# B&R Automation Studio project TD52 (part 92)

### sPLC.var - SAFETY PLC variables
```iecst
VAR
	bSafeIN_ECW_PumpsOFF : BOOL := FALSE; (*To SafetyPLC - No engine cooling water pump is running*)
	bSafeIN_EO_PumpsOFF : BOOL := FALSE; (*To SafetyPLC - No engine oil pump is running*)
	bSafeIN_ERV_ColdCountry : BOOL := FALSE; (*To SafetyPLC - Cold country mode is active*)
	bSafeIN_ERV_Lou_PC_CL : BOOL := FALSE; (*To SafetyPLC - Plausibility check for closing the louvres*)
	bSafeIN_ERV_Lou_PC_OP : BOOL := FALSE; (*To SafetyPLC - Plausibility check for opening the louvres*)
	bSafeIN_Reset_sPLC : BOOL := FALSE; (*To SafetyPLC - RESET - Release sDOs - Reset IO card failures*)
	bSafeModuleOK_101 : BOOL := FALSE; (*Safe communication channel - Node 101 OK*)
	bSafeModuleOK_102 : BOOL := FALSE; (*Safe communication channel - Node 102 OK*)
	bSafeModuleOK_103 : BOOL := FALSE; (*Safe communication channel - Node 103 OK*)
	bSafeModuleOK_104 : BOOL := FALSE; (*Safe communication channel - Node 104 OK*)
	bSafeModuleOK_105 : BOOL := FALSE; (*Safe communication channel - Node 105 OK*)
	bSafeModuleOK_201 : BOOL := FALSE; (*Safe communication channel - Node 201 OK*)
	bSafeModuleOK_202 : BOOL := FALSE; (*Safe communication channel - Node 202 OK*)
	bSafeModuleOK_203 : BOOL := FALSE; (*Safe communication channel - Node 203 OK*)
	bSafeModuleOK_204 : BOOL := FALSE; (*Safe communication channel - Node 204 OK*)
	bSafeModuleOK_205 : BOOL := FALSE; (*Safe communication channel - Node 205 OK*)
	bSafeModuleOK_206 : BOOL := FALSE; (*Safe communication channel - Node 206 OK*)
	bSafeModuleOK_207 : BOOL := FALSE; (*Safe communication channel - Node 207 OK*)
	bSafeModuleOK_208 : BOOL := FALSE; (*Safe communication channel - Node 208 OK*)
	bSafeModuleOK_209 : BOOL := FALSE; (*Safe communication channel - Node 209 OK*)
	bSafeModuleOK_210 : BOOL := FALSE; (*Safe communication channel - Node 210 OK*)
	bSafeModuleOK_300 : BOOL := FALSE; (*Safe communication channel - Node 300 OK*)
	bSafeModuleOK_301 : BOOL := FALSE; (*Safe communication channel - Node 301 OK*)
	bSafeOUT_F01_N_DiffOK : BOOL := FALSE; (*From SafetyPLC - Function 01 - Speed difference OK*)
	bSafeOUT_F01_N_Nom90 : BOOL := FALSE; (*From SafetyPLC - Function 01 - Actual engine speed >= 90% of nominal speed*)
	bSafeOUT_F01_OK : BOOL := FALSE; (*From SafetyPLC - Function 01 - Speed measurement OK*)
	bSafeOUT_F02_OK : BOOL := FALSE; (*From SafetyPLC - Function 02 - Ignition is operating*)
	bSafeOUT_F02_OK_PC : BOOL := FALSE; (*From SafetyPLC - Function 02 - Ignition plausibility check - OK*)
	bSafeOUT_F03_OK : BOOL := FALSE; (*From SafetyPLC - Function 03 - Oil pressure MIN OK*)
	bSafeOUT_F03_Pr_EO_DiffOK : BOOL := FALSE; (*From SafetyPLC - Function 03 - Oil pressure difference OK*)
	bSafeOUT_F04_OK : BOOL := FALSE; (*From SafetyPLC - Function 04 - Oil pressure MAX OK*)
	bSafeOUT_F05_OK : BOOL := FALSE; (*From SafetyPLC - Function 05 - Engine cooling water pressure MIN OK*)
	bSafeOUT_F05_Pr_ECW_DiffOK : BOOL := FALSE; (*From SafetyPLC - Function 05 - Engine cooling water pressure difference OK*)
	bSafeOUT_F06_OK : BOOL := FALSE; (*From SafetyPLC - Function 06 - Engine cooling water pressure MAX OK*)
	bSafeOUT_F07_GCB_RUC : BOOL := FALSE; (*From SafetyPLC - Function 07 - GCB - Release undervoltage coil OK*)
	bSafeOUT_F07_GCB_RUC_PS : BOOL := FALSE; (*From SafetyPLC - Function 07 - GCB - Release undervoltage coil OK - Physical state*)
	bSafeOUT_F07_OK : BOOL := FALSE; (*From SafetyPLC - Function 07 - Grid disconnection OK*)
	bSafeOUT_F07_Rel_Sync_Load : BOOL := FALSE; (*From SafetyPLC - Function 07 - Release synchronizing and load OK*)
	bSafeOUT_F07_Rel_Sync_Load_PS : BOOL := FALSE; (*From SafetyPLC - Function 07 - Release synchronizing and load - Physical state*)
	bSafeOUT_F08_GenPrctTrip_OK : BOOL := FALSE; (*From SafetyPLC - Function 08 - Generator protection trip OK*)
	bSafeOUT_F08_OlShortCirc_OK : BOOL := FALSE; (*From SafetyPLC - Function 08 - Generator overload/short circuit OK*)
	bSafeOUT_F09_Cust_OK : BOOL := FALSE; (*From SafetyPLC - Function 09 - Room ventilation operating*)
	bSafeOUT_F09_Cust_OK_PC : BOOL := FALSE; (*From SafetyPLC - Function 09 - Room ventilation plausibility check OK*)
	bSafeOUT_F09_DI_ERV_Cust : BOOL := FALSE; (*From SafetyPLC - Function 09 - Room ventilation operating - Digital input*)
	bSafeOUT_F09_Door_OK : BOOL := FALSE; (*From SafetyPLC - Function 09 - Doors closed*)
	bSafeOUT_F09_ERV_PC_Forced : BOOL := FALSE; (*From SafetyPLC - Function 09 - Forced ERV plausibility checks*)
	bSafeOUT_F09_INL1_Fan_OK : BOOL := FALSE; (*From SafetyPLC - Function 09 - Group 1 - Inlet air fan operating*)
	bSafeOUT_F09_INL1_Fan_OK_PC : BOOL := FALSE; (*From SafetyPLC - Function 09 - Group 1 - Inlet air fan plausibility check OK*)
	bSafeOUT_F09_INL1_Lou_OK : BOOL := FALSE; (*From SafetyPLC - Function 09 - Group 1 - Inlet air louvre OK*)
	bSafeOUT_F09_INL1_Lou_OK_PC : BOOL := FALSE; (*From SafetyPLC - Function 09 - Group 1 - Inlet air louvre plausibility check OK*)
	bSafeOUT_F09_INL2_Fan_OK : BOOL := FALSE; (*From SafetyPLC - Function 09 - Group 2 - Inlet air fan operating*)
	bSafeOUT_F09_INL2_Fan_OK_PC : BOOL := FALSE; (*From SafetyPLC - Function 09 - Group 2 - Inlet air fan plausibility check OK*)
	bSafeOUT_F09_INL2_Lou_OK : BOOL := FALSE; (*From SafetyPLC - Function 09 - Group 2 - Inlet air louvre OK*)
	bSafeOUT_F09_INL2_Lou_OK_PC : BOOL := FALSE; (*From SafetyPLC - Function 09 - Group 2 - Inlet air louvre plausibility check OK*)
	bSafeOUT_F09_INL3_Fan_OK : BOOL := FALSE; (*From SafetyPLC - Function 09 - Group 3 - Inlet air fan operating*)
	bSafeOUT_F09_INL3_Fan_OK_PC : BOOL := FALSE; (*From SafetyPLC - Function 09 - Group 3 - Inlet air fan plausibility check OK*)
	bSafeOUT_F09_INL3_Lou_OK : BOOL := FALSE; (*From SafetyPLC - Function 09 - Group 3 - Inlet air louvre OK*)
	bSafeOUT_F09_INL3_Lou_OK_PC : BOOL := FALSE; (*From SafetyPLC - Function 09 - Group 3 - Inlet air louvre plausibility check OK*)
	bSafeOUT_F09_INL4_Fan_OK : BOOL := FALSE; (*From SafetyPLC - Function 09 - Group 4 - Inlet air fan operating*)
	bSafeOUT_F09_INL4_Fan_OK_PC : BOOL := FALSE; (*From SafetyPLC - Function 09 - Group 4 - Inlet air fan plausibility check OK*)
	bSafeOUT_F09_INL4_Lou_OK : BOOL := FALSE; (*From SafetyPLC - Function 09 - Group 4 - Inlet air louvre OK*)
	bSafeOUT_F09_INL4_Lou_OK_PC : BOOL := FALSE; (*From SafetyPLC - Function 09 - Group 4 - Inlet air louvre plausibility check OK*)
	bSafeOUT_F09_INL5_Fan_OK : BOOL := FALSE; (*From SafetyPLC - Function 09 - Group 5 - Inlet air fan operating*)
	bSafeOUT_F09_INL5_Fan_OK_PC : BOOL := FALSE; (*From SafetyPLC - Function 09 - Group 5 - Inlet air fan plausibility check OK*)
	bSafeOUT_F09_INL5_Lou_OK : BOOL := FALSE; (*From SafetyPLC - Function 09 - Group 5 - Inlet air louvre OK*)
	bSafeOUT_F09_INL5_Lou_OK_PC : BOOL := FALSE; (*From SafetyPLC - Function 09 - Group 5 - Inlet air louvre plausibility check OK*)
	bSafeOUT_F09_INL6_Fan_OK : BOOL := FALSE; (*From SafetyPLC - Function 09 - Group 6 - Inlet air fan operating*)
	bSafeOUT_F09_INL6_Fan_OK_PC : BOOL := FALSE; (*From SafetyPLC - Function 09 - Group 6 - Inlet air fan plausibility check OK*)
	bSafeOUT_F09_INL6_Lou_OK : BOOL := FALSE; (*From SafetyPLC - Function 09 - Group 6 - Inlet air louvre OK*)
	bSafeOUT_F09_INL6_Lou_OK_PC : BOOL := FALSE; (*From SafetyPLC - Function 09 - Group 6 - Inlet air louvre plausibility check OK*)
	bSafeOUT_F09_OTL1_Lou_OK : BOOL := FALSE; (*From SafetyPLC - Function 09 - Group 1 - Outlet air louvre OK*)
	bSafeOUT_F09_OTL1_Lou_OK_PC : BOOL := FALSE; (*From SafetyPLC - Function 09 - Group 1 - Outlet air louvre plausibility check OK*)
	bSafeOUT_F09_OTL2_Lou_OK : BOOL := FALSE; (*From SafetyPLC - Function 09 - Group 2 - Outlet air louvre OK*)
	bSafeOUT_F09_OTL2_Lou_OK_PC : BOOL := FALSE; (*From SafetyPLC - Function 09 - Group 2 - Outlet air louvre plausibility check OK*)
	bSafeOUT_F09_OTL3_Lou_OK : BOOL := FALSE; (*From SafetyPLC - Function 09 - Group 3 - Outlet air louvre OK*)
	bSafeOUT_F09_OTL3_Lou_OK_PC : BOOL := FALSE; (*From SafetyPLC - Function 09 - Group 3 - Outlet air louvre plausibility check OK*)
	bSafeOUT_F09_OTL4_Lou_OK : BOOL := FALSE; (*From SafetyPLC - Function 09 - Group 4 - Outlet air louvre OK*)
	bSafeOUT_F09_OTL4_Lou_OK_PC : BOOL := FALSE; (*From SafetyPLC - Function 09 - Group 4 - Outlet air louvre plausibility check OK*)
	bSafeOUT_F09_OTL5_Lou_OK : BOOL := FALSE; (*From SafetyPLC - Function 09 - Group 5 - Outlet air louvre OK*)
	bSafeOUT_F09_OTL5_Lou_OK_PC : BOOL := FALSE; (*From SafetyPLC - Function 09 - Group 5 - Outlet air louvre plausibility check OK*)
	bSafeOUT_F09_OTL6_Lou_OK : BOOL := FALSE; (*From SafetyPLC - Function 09 - Group 6 - Outlet air louvre OK*)
	bSafeOUT_F09_OTL6_Lou_OK_PC : BOOL := FALSE; (*From SafetyPLC - Function 09 - Group 6 - Outlet air louvre plausibility check OK*)
	bSafeOUT_F10_DO_EmStop : BOOL := FALSE; (*From SafetyPLC - Function 10 - DO Emergency stop signalling*)
	bSafeOUT_F10_DO_EmStop_PS : BOOL := FALSE; (*From SafetyPLC - Function 10 - DO Emergency stop signalling - Physical state*)
	bSafeOUT_F10_EmStop_M_OK : BOOL := FALSE; (*From SafetyPLC - Function 10 - Emergency stop push button - Module interface panel*)
	bSafeOUT_F10_EmStop_OK : BOOL := FALSE; (*From SafetyPLC - Function 10 - Emergency stop push button*)
	bSafeOUT_F10_SafetyLoop_EmStop : BOOL := FALSE; (*From SafetyPLC - Function 10 - Safety loop - Emergency stop push button OK*)
	bSafeOUT_F11_SafetyLoop_A1_OK : BOOL := FALSE; (*From SafetyPLC - Function 11 - Safety loop 1 - module control panel OK*)
	bSafeOUT_F11_SafetyLoop_A2_OK : BOOL := FALSE; (*From SafetyPLC - Function 11 - Safety loop 2 - module control panel OK*)
	bSafeOUT_F11_SafetyLoop_M_OK : BOOL := FALSE; (*From SafetyPLC - Function 11 - Safety loop - module interface panel OK*)
	bSafeOUT_F12_DCGA_OK : BOOL := FALSE; (*From SafetyPLC - Function 12 - Gas supply interruption OK - DCGA (Decentral gas addition)*)
	bSafeOUT_F12_DCGA_SD_Dem : BOOL := FALSE; (*From SafetyPLC - Function 12 - Demand gas safety device - DCGA*)
	bSafeOUT_F12_DCGA_SD_Dem_PS : BOOL := FALSE; (*From SafetyPLC - Function 12 - Demand gas safety device - DCGA - Physical state*)
	bSafeOUT_F12_DI_DCGA_SafeDevOK : BOOL := FALSE; (*From SafetyPLC - Function 12 - Digital Input - Gas safety device OK - DCGA*)
	bSafeOUT_F12_DI_GT1_SafeDevOK : BOOL := FALSE; (*From SafetyPLC - Function 12 - Digital Input - Gas safety device OK - Gastrain 1*)
	bSafeOUT_F12_DI_GT2_SafeDevOK : BOOL := FALSE; (*From SafetyPLC - Function 12 - Digital Input - Gas safety device OK - Gastrain 2*)
	bSafeOUT_F12_DI_GT3_SafeDevOK : BOOL := FALSE; (*From SafetyPLC - Function 12 - Digital Input - Gas safety device OK - Gastrain 3*)
	bSafeOUT_F12_DI_GT4_SafeDevOK : BOOL := FALSE; (*From SafetyPLC - Function 12 - Digital Input - Gas safety device OK - Gastrain 4*)
	bSafeOUT_F12_GT1_OK : BOOL := FALSE; (*From SafetyPLC - Function 12 - Gas supply interruption OK - Gas train 1*)
	bSafeOUT_F12_GT1_SD_Dem : BOOL := FALSE; (*From SafetyPLC - Function 12 - Demand gas safety device - Gastrain 1*)
	bSafeOUT_F12_GT1_SD_Dem_PS : BOOL := FALSE; (*From SafetyPLC - Function 12 - Demand gas safety device - Gastrain 1 - Physical state*)
	bSafeOUT_F12_GT2_OK : BOOL := FALSE; (*From SafetyPLC - Function 12 - Gas supply interruption OK - Gas train 2*)
	bSafeOUT_F12_GT2_SD_Dem : BOOL := FALSE; (*From SafetyPLC - Function 12 - Demand gas safety device - Gastrain 2*)
	bSafeOUT_F12_GT2_SD_Dem_PS : BOOL := FALSE; (*From SafetyPLC - Function 12 - Demand gas safety device - Gastrain 2 - Physical state*)
	bSafeOUT_F12_GT3_OK : BOOL := FALSE; (*From SafetyPLC - Function 12 - Gas supply interruption OK - Gas train 3*)
	bSafeOUT_F12_GT3_SD_Dem : BOOL := FALSE; (*From SafetyPLC - Function 12 - Demand gas safety device - Gastrain 3*)
	bSafeOUT_F12_GT3_SD_Dem_PS : BOOL := FALSE; (*From SafetyPLC - Function 12 - Demand gas safety device - Gastrain 3 - Physical state*)
	bSafeOUT_F12_GT4_OK : BOOL := FALSE; (*From SafetyPLC - Function 12 - Gas supply interruption OK - Gas train 4*)
	bSafeOUT_F12_GT4_SD_Dem : BOOL := FALSE; (*From SafetyPLC - Function 12 - Demand gas safety device - Gastrain 4*)
	bSafeOUT_F12_GT4_SD_Dem_PS : BOOL := FALSE; (*From SafetyPLC - Function 12 - Demand gas safety device - Gastrain 4 - Physical state*)
	bSafeOUT_F12_Rel_GV1 : BOOL := FALSE; (*From SafetyPLC - Function 12 - Gas valves from gas train 1 released*)
	bSafeOUT_F12_Rel_GV1a_PS : BOOL := FALSE; (*From SafetyPLC - Function 12 - Gas valve 1a - Physical state*)
	bSafeOUT_F12_Rel_GV1b_PS : BOOL := FALSE; (*From SafetyPLC - Function 12 - Gas valve 1b - Physical state*)
	bSafeOUT_F12_Rel_GV2 : BOOL := FALSE; (*From SafetyPLC - Function 12 - Gas valves from gas train 2 released*)
	bSafeOUT_F12_Rel_GV2a_PS : BOOL := FALSE; (*From SafetyPLC - Function 12 - Gas valve 2a - Physical state*)
	bSafeOUT_F12_Rel_GV2b_PS : BOOL := FALSE; (*From SafetyPLC - Function 12 - Gas valve 2b - Physical state*)
	bSafeOUT_F12_Rel_GV3 : BOOL := FALSE; (*From SafetyPLC - Function 12 - Gas valves from gas train 3 released*)
	bSafeOUT_F12_Rel_GV3a_PS : BOOL := FALSE; (*From SafetyPLC - Function 12 - Gas valve 3a - Physical state*)
	bSafeOUT_F12_Rel_GV3b_PS : BOOL := FALSE; (*From SafetyPLC - Function 12 - Gas valve 3b - Physical state*)
	bSafeOUT_F12_Rel_GV4 : BOOL := FALSE; (*From SafetyPLC - Function 12 - Gas valves from gas train 4 released*)
	bSafeOUT_F12_Rel_GV4a_PS : BOOL := FALSE; (*From SafetyPLC - Function 12 - Gas valve 4a - Physical state*)
	bSafeOUT_F12_Rel_GV4b_PS : BOOL := FALSE; (*From SafetyPLC - Function 12 - Gas valve 4b - Physical state*)
	bSafeOUT_F12_Rel_GVa_DCGA_PS : BOOL := FALSE; (*From SafetyPLC - Function 12 - Gas valve a for DCGA - Physical state*)
	bSafeOUT_F12_Rel_GVb_DCGA_PS : BOOL := FALSE; (*From SafetyPLC - Function 12 - Gas valve b for DCGA - Physical state*)
	bSafeOUT_F12_Rel_GV_DCGA : BOOL := FALSE; (*From SafetyPLC - Function 12 - Gas valves from DCGA released*)
	bSafeOUT_F16_DI_ScavFlapClosed : BOOL := FALSE; (*From SafetyPLC - Function 20 - Scavenging flap closed OK*)
	bSafeOUT_F16_ScavFlapPos_OK : BOOL := FALSE; (*From SafetyPLC - Function 20 - Scavenging flap position OK*)
	bSafeOUT_F16_ScavFlapPos_OK_PC : BOOL := FALSE; (*From SafetyPLC - Function 20 - Scavenging flap position - plausibility check  OK*)
	bSafeOUT_F16_TS_ScavFlap_OK : BOOL := FALSE; (*From SafetyPLC - Function 20 - Scavenging flap temperature switch  OK*)
	bSafeOUT_F17_Purge_OK : BOOL := FALSE; (*From SafetyPLC - Function 17 - Purge state OK*)
	bSafeOUT_F20_FS_HWHT_Lo_DI : BOOL := FALSE; (*From SafetyPLC - Function 20 - High temperature heating water flow minimum - DI OK*)
	bSafeOUT_F20_FS_HWHT_Lo_OK : BOOL := FALSE; (*From SafetyPLC - Function 20 - High temperature heating water flow minimum OK*)
	bSafeOUT_F20_FS_HWHT_Lo_OK_PC : BOOL := FALSE; (*From SafetyPLC - Function 20 - High temperature heating water flow minimum - plausibility check OK*)
	bSafeOUT_F20_FS_HWLT_Lo_DI : BOOL := FALSE; (*From SafetyPLC - Function 20 - Low temperature heating water flow minimum - DI OK*)
	bSafeOUT_F20_FS_HWLT_Lo_OK : BOOL := FALSE; (*From SafetyPLC - Function 20 - Low temperature heating water flow minimum OK*)
	bSafeOUT_F20_FS_HWLT_Lo_OK_PC : BOOL := FALSE; (*From SafetyPLC - Function 20 - Low temperature heating water flow minimum - plausibility check OK*)
	bSafeOUT_F20_HWcirc_Cust_OK : BOOL := FALSE; (*From SafetyPLC - Function 20 - Customer heating water circuit OK*)
	bSafeOUT_F20_LS_HWHT_Lo_OK : BOOL := FALSE; (*From SafetyPLC - Function 20 - High temperature heating water level minimum OK*)
	bSafeOUT_F20_LS_HWLT_Lo_OK : BOOL := FALSE; (*From SafetyPLC - Function 20 - Low temperature heating water level minimum OK*)
	bSafeOUT_F20_PS1_HWHT_Hi_OK : BOOL := FALSE; (*From SafetyPLC - Function 20 - High temperature heating water pressure 1 maximum OK*)
	bSafeOUT_F20_PS1_HWHT_Lo_DI : BOOL := FALSE; (*From SafetyPLC - Function 20 - High temperature heating water pressure 1 minimum - DI OK*)
	bSafeOUT_F20_PS1_HWHT_Lo_OK : BOOL := FALSE; (*From SafetyPLC - Function 20 - High temperature heating water pressure 1 minimum OK*)
	bSafeOUT_F20_PS1_HWLT_Hi_OK : BOOL := FALSE; (*From SafetyPLC - Function 20 - Low temperature heating water pressure 1 maximum OK*)
	bSafeOUT_F20_PS1_HWLT_Lo_DI : BOOL := FALSE; (*From SafetyPLC - Function 20 - Low temperature heating water pressure 1 minimum - DI OK*)
	bSafeOUT_F20_PS1_HWLT_Lo_OK : BOOL := FALSE; (*From SafetyPLC - Function 20 - Low temperature heating water pressure 1 minimum OK*)
	bSafeOUT_F20_PS2_HWHT_Hi_OK : BOOL := FALSE; (*From SafetyPLC - Function 20 - High temperature heating water pressure 2 maximum OK*)
	bSafeOUT_F20_PS2_HWHT_Lo_DI : BOOL := FALSE; (*From SafetyPLC - Function 20 - High temperature heating water pressure 2 minimum - DI OK*)
	bSafeOUT_F20_PS2_HWHT_Lo_OK : BOOL := FALSE; (*From SafetyPLC - Function 20 - High temperature heating water pressure 2 minimum OK*)
	bSafeOUT_F20_PS2_HWLT_Hi_OK : BOOL := FALSE; (*From SafetyPLC - Function 20 - Low temperature heating water pressure 2 maximum OK*)
	bSafeOUT_F20_PS2_HWLT_Lo_DI : BOOL := FALSE; (*From SafetyPLC - Function 20 - Low temperature heating water pressure 2 minimum - DI OK*)
	bSafeOUT_F20_PS2_HWLT_Lo_OK : BOOL := FALSE; (*From SafetyPLC - Function 20 - Low temperature heating water pressure 2 minimum OK*)
	bSafeOUT_F20_TS1_HWHT_Hi_OK : BOOL := FALSE; (*From SafetyPLC - Function 20 - High temperature heating water temperature 1 maximum OK*)
	bSafeOUT_F20_TS1_HWLT_Hi_OK : BOOL := FALSE; (*From SafetyPLC - Function 20 - Low temperature heating water temperature 1 maximum OK*)
	bSafeOUT_F20_TS2_HWHT_Hi_OK : BOOL := FALSE; (*From SafetyPLC - Function 20 - High temperature heating water temperature 2 maximum OK*)
	bSafeOUT_F20_TS2_HWLT_Hi_OK : BOOL := FALSE; (*From SafetyPLC - Function 20 - Low temperature heating water temperature 2 maximum OK*)
	bSafeOUT_F21_Pr_EG_Hi_OK : BOOL := FALSE; (*From SafetyPLC - Function 20 - Exhaust gas backpressure high OK*)
	bSafeOUT_F99_Rel_SF_OK : BOOL := FALSE; (*From SafetyPLC - Function 99 - Release safety functions OK*)
	bSafeOUT_F99_Rel_SF_OK_A_PS : BOOL := FALSE; (*From SafetyPLC - Function 99 - Release safety functions - Module control panel - Physical state*)
	bSafeOUT_F99_Rel_SF_OK_M_PS : BOOL := FALSE; (*From SafetyPLC - Function 99 - Release safety functions - Module interface panel - Physical state*)
	bSafeOUT_F99_SafetyLoop_Eng : BOOL := FALSE; (*From SafetyPLC - Function 10 - Safety loop - Engine OK*)
	iParaRead_sPLC : ARRAY[0..29] OF UINT := [30(0)]; (*Read Parameter from SafetyPLC*)
	iSafeIN_Eng_Motortype : INT := 0; (*To SafetyPLC - Para: Motortype*)
	iSafeIN_N_EngAct : INT := 0; (*To SafetyPLC - Actual engine speed [rpm]*)
	iSafeIN_N_EngNom : INT := 0; (*To SafetyPLC - Para: Engine nominal speed [rpm]*)
	iSafeOUT_F01_N_EngAct : DINT := 0; (*From SafetyPLC - Function 01 - Actual engine speed [rpm]*)
	iSafeOUT_F01_N_EngAct_Diff : DINT := 0; (*From SafetyPLC - Function 01 - Speed difference [rpm]*)
	iSafeOUT_F01_N_Nom90_10s_ET : DINT := 0; (*From SafetyPLC - Function 01 - Speed >= 90% of nominal speed - Elipsed time*)
	iSafeOUT_F01_SDC_30s_ET : DINT := 0; (*From SafetyPLC - Function 01 - Speed difference check - Elipsed time*)
	iSafeOUT_F01_Standstill_1m_ET : DINT := 0; (*From SafetyPLC - Function 01 - Speed < 80rpm - Elipsed time*)
	iSafeOUT_F03_Pr_EO : DINT := 0; (*From SafetyPLC - Function 03 - Actual oil pressure at last lubrication point [mbar]*)
	iSafeOUT_F03_Pr_EO_Diff : DINT := 0; (*From SafetyPLC - Function 03 - Oil pressure difference [mbar]*)
	iSafeOUT_F03_Pr_EO_Fr_1m_ET : DINT := 0; (*From SafetyPLC - Function 03 - Oil pressure frozen - Elipsed time*)
	iSafeOUT_F03_Pr_EO_Standstill : DINT := 0; (*From SafetyPLC - Function 03 - Oil pressure at last lubrication point - At standstill [mbar]*)
	iSafeOUT_F04_EO_PumpsOff_2m_ET : DINT := 0; (*From SafetyPLC - Function 04 - Oil pumps off for 120s - Elipsed time*)
	iSafeOUT_F04_Pr_EOaP : DINT := 0; (*From SafetyPLC - Function 04 - Actual oil pressure after pump [mbar]*)
	iSafeOUT_F04_Pr_EOaP_Fr_1m_ET : DINT := 0; (*From SafetyPLC - Function 04 - Oil pressure after pump frozen - Elipsed time*)
	iSafeOUT_F04_Pr_EOaP_Standstill : DINT := 0; (*From SafetyPLC - Function 04 - Oil pressure after pump - At standstill [mbar]*)
	iSafeOUT_F05_Pr_ECW : DINT := 0; (*From SafetyPLC - Function 05 - Actual engine cooling water pressure [mbar]*)
	iSafeOUT_F05_Pr_ECW_Diff : DINT := 0; (*From SafetyPLC - Function 05 - Engine cooling water pressure difference [mbar]*)
	iSafeOUT_F05_Pr_ECW_Fr_1m_ET : DINT := 0; (*From SafetyPLC - Function 05 - Engine cooling water pressure frozen - Elipsed time*)
	iSafeOUT_F06_ECW_PumpsOff_2m_ET : DINT := 0; (*From SafetyPLC - Function 06 - Engine cooling water pumps off for 120s - Elipsed time*)
	iSafeOUT_F06_Pr_ECWaP : DINT := 0; (*From SafetyPLC - Function 06 - Actual engine cooling water pressure after pump [mbar]*)
	iSafeOUT_F06_Pr_ECWaP_Fr_1m_ET : DINT := 0; (*From SafetyPLC - Function 06 - Engine cooling water pressure after pump frozen - Elipsed time*)
	iSafeOUT_F07_GCB_On_10s_ET : DINT := 0; (*From SafetyPLC - Function 07 - Generator circuit breaker ON for 10s - Elipsed time*)
	iSafeOUT_F07_GCB_On_60s_ET : DINT := 0; (*From SafetyPLC - Function 07 - Generator circuit breaker ON for 60s - Elipsed time*)
	iSafeOUT_F09_CRC : UDINT := 0; (*From SafetyPLC - Function 09 - Ventilation - CRC*)
	iSafeOUT_F09_Cust_OK_15s_ET : DINT := 0; (*From SafetyPLC - Function 09 - Room ventilation not operating - Elapsed time*)
	iSafeOUT_F09_Cust_PC_ET : DINT := 0; (*From SafetyPLC - Function 09 - Room ventilation plausibility check - Elapsed time*)
	iSafeOUT_F09_Door_OK_15s_ET : DINT := 0; (*From SafetyPLC - Function 09 - Doors not closed - Elapsed time*)
	iSafeOUT_F09_INL1_Fan_OK_1m_ET : DINT := 0; (*From SafetyPLC - Function 09 - Group 1 - Inlet air fan not operating - Elapsed time*)
	iSafeOUT_F09_INL1_Lou_OK_1m_ET : DINT := 0; (*From SafetyPLC - Function 09 - Group 1 - Inlet air louvre not OK - Elapsed time*)
	iSafeOUT_F09_INL2_Fan_OK_1m_ET : DINT := 0; (*From SafetyPLC - Function 09 - Group 2 - Inlet air fan not operating - Elapsed time*)
	iSafeOUT_F09_INL2_Lou_OK_1m_ET : DINT := 0; (*From SafetyPLC - Function 09 - Group 2 - Inlet air louvre not OK - Elapsed time*)
	iSafeOUT_F09_INL3_Fan_OK_1m_ET : DINT := 0; (*From SafetyPLC - Function 09 - Group 3 - Inlet air fan not operating - Elapsed time*)
	iSafeOUT_F09_INL3_Lou_OK_1m_ET : DINT := 0; (*From SafetyPLC - Function 09 - Group 3 - Inlet air louvre not OK - Elapsed time*)
	iSafeOUT_F09_INL4_Fan_OK_1m_ET : DINT := 0; (*From SafetyPLC - Function 09 - Group 4 - Inlet air fan not operating - Elapsed time*)
	iSafeOUT_F09_INL4_Lou_OK_1m_ET : DINT := 0; (*From SafetyPLC - Function 09 - Group 4 - Inlet air louvre not OK - Elapsed time*)
	iSafeOUT_F09_INL5_Fan_OK_1m_ET : DINT := 0; (*From SafetyPLC - Function 09 - Group 5 - Inlet air fan not operating - Elapsed time*)
	iSafeOUT_F09_INL5_Lou_OK_1m_ET : DINT := 0; (*From SafetyPLC - Function 09 - Group 5 - Inlet air louvre not OK - Elapsed time*)
	iSafeOUT_F09_INL6_Fan_OK_1m_ET : DINT := 0; (*From SafetyPLC - Function 09 - Group 6 - Inlet air fan not operating - Elapsed time*)
	iSafeOUT_F09_INL6_Lou_OK_1m_ET : DINT := 0; (*From SafetyPLC - Function 09 - Group 6 - Inlet air louvre not OK - Elapsed time*)
	iSafeOUT_F09_Nr_PC_NotDone : INT := 0; (*From SafetyPLC - Function 09 - Number of plausibility checks not performed*)
	iSafeOUT_F09_OTL1_Lou_OK_1m_ET : DINT := 0; (*From SafetyPLC - Function 09 - Group 1 - Outlet air louvre not OK - Elapsed time*)
	iSafeOUT_F09_OTL2_Lou_OK_1m_ET : DINT := 0; (*From SafetyPLC - Function 09 - Group 2 - Outlet air louvre not OK - Elapsed time*)
	iSafeOUT_F09_OTL3_Lou_OK_1m_ET : DINT := 0; (*From SafetyPLC - Function 09 - Group 3 - Outlet air louvre not OK - Elapsed time*)
	iSafeOUT_F09_OTL4_Lou_OK_1m_ET : DINT := 0; (*From SafetyPLC - Function 09 - Group 4 - Outlet air louvre not OK - Elapsed time*)
	iSafeOUT_F09_OTL5_Lou_OK_1m_ET : DINT := 0; (*From SafetyPLC - Function 09 - Group 5 - Outlet air louvre not OK - Elapsed time*)
	iSafeOUT_F09_OTL6_Lou_OK_1m_ET : DINT := 0; (*From SafetyPLC - Function 09 - Group 6 - Outlet air louvre not OK - Elapsed time*)
	iSafeOUT_F12_DCGA_LC_130s_ET : DINT := 0; (*From SafetyPLC - Function 12 - DCGA - Gas leakage check 130s - Elipsed time*)
	iSafeOUT_F12_GT1_LC_130s_ET : DINT := 0; (*From SafetyPLC - Function 12 - Gas train 1 - Gas leakage check 130s - Elipsed time*)
	iSafeOUT_F12_GT2_LC_130s_ET : DINT := 0; (*From SafetyPLC - Function 12 - Gas train 2 - Gas leakage check 130s - Elipsed time*)
	iSafeOUT_F12_GT3_LC_130s_ET : DINT := 0; (*From SafetyPLC - Function 12 - Gas train 3 - Gas leakage check 130s - Elipsed time*)
	iSafeOUT_F12_GT4_LC_130s_ET : DINT := 0; (*From SafetyPLC - Function 12 - Gas train 4 - Gas leakage check 130s - Elipsed time*)
	iSafeOUT_F12_GV_Open_60s_ET : DINT := 0; (*From SafetyPLC - Function 12 - Gas valves open for 60s - Elipsed time*)
	iSafeOUT_F16_ScavFlapPos_PC_ET : DINT := 0; (*From SafetyPLC - Function 16 - Scavenging flap position - plausibility check - Elipsed time OK*)
	iSafeOUT_F17_Vol_PurgeAir : DINT := 0; (*From SafetyPLC - Function 17 - Purge air volume [l]*)
	iSafeOUT_F20_CRC : UDINT := 0; (*From SafetyPLC - Function 20 - Heating water - CRC*)
	iSafeOUT_F20_FS_HWHT_Lo_OK_ET : DINT := 0; (*From SafetyPLC - Function 20 - High temperature heating water flow minimum - Elipsed time OK*)
	iSafeOUT_F20_FS_HWHT_Lo_PC_ET : DINT := 0; (*From SafetyPLC - Function 20 - High temperature heating water flow minimum - plausibility check - Elipsed time OK*)
	iSafeOUT_F20_FS_HWLT_Lo_OK_ET : DINT := 0; (*From SafetyPLC - Function 20 - Low temperature heating water flow minimum - Elipsed time OK*)
	iSafeOUT_F20_FS_HWLT_Lo_PC_ET : DINT := 0; (*From SafetyPLC - Function 20 - Low temperature heating water flow minimum - plausibility check - Elipsed time OK*)
	iSafeOUT_F20_PS1_HWHT_Lo_OK_ET : DINT := 0; (*From SafetyPLC - Function 20 - High temperature heating water pressure 1 minimum - Elipsed time OK*)
	iSafeOUT_F20_PS1_HWLT_Lo_OK_ET : DINT := 0; (*From SafetyPLC - Function 20 - Low temperature heating water pressure 1 minimum - Elipsed time OK*)
	iSafeOUT_F20_PS2_HWHT_Lo_OK_ET : DINT := 0; (*From SafetyPLC - Function 20 - High temperature heating water pressure 2 minimum - Elipsed time OK*)
	iSafeOUT_F20_PS2_HWLT_Lo_OK_ET : DINT := 0; (*From SafetyPLC - Function 20 - Low temperature heating water pressure 2 minimum - Elipsed time OK*)
	iSafeOUT_FwVers_sPLC : UDINT := 0; (*From SafetyPLC - Actual firmware version*)
	MM2VIS_sPLC : MM2VIS_sPLC_Struct;
	VIS2MM_sPLC : VIS2MM_sPLC_struct;
END_VAR
```

### Program Logical/EngineGeneral/GeneralEG (IEC, version 4.10.0) - general functions

#### GeneralEGCyclic.st - Cyclic code
```iecst
(*******************************************************************************
GeneralEG		general functions

This code is confidential and proprietary to the INNIO Company.
It may not be used in any form, or reproduced in any manner,
without the express written permission of the INNIO Company.
Copyright, INNIO Company, 2021

Customized modifications: -
------------------------

History:
-------
V03.99.00.00	08.02.2013 	Tinello 	Created
V04.03.00.00	20.01.2016	Tinello		Release Module if ParaSetupOk = TRUE added
V04.05.00.00	26.01.2017	Tinello		Release Module from 10s -> 20s
V04.10.00.00	28.01.2021	Tinello		operation mode added

(*******************************************************************************)
PROGRAM _CYCLIC

	(* Release Module if ParaSetupOk = TRUE *)
	xTON_ParaSetupOk(IN		:= IN_EG.tPB2MM.bParaSetupOk, PT:= T#20s);
	bRelModul_ParaSetupOk	:= xTON_ParaSetupOk.Q;

	(* Engine motortype *)
	xEngType.Motortype 	:= INT_TO_UINT(Para.iEng_Motortype);
	xEngType();

	(* Number of cylinder --> VISU *)
	MM2VIS.iNum_Cyl 	:= xEngType.NumberOfCylinder;

	(* engine start speed reached *)
	xGR_MAXR_StartSpd(In:= IN_EG.rN_EngAct,   Gw := Para.rN_EngStart_LimHi, Hy := Para.rN_EngStart_HyHi);
	xTOF_StartSpd(IN 	:= xGR_MAXR_StartSpd.Q AND bRelModul_ParaSetupOk, 	PT := T#10s);
	bStartSpd			:= xTOF_StartSpd.Q;

	(* Power signal missing *)
	xGR_MINR_P_Lo(In 	:= IN_EG.rP_Act_Norm, Gw := Para.rP_LimLo, Hy := Para.rP_HyLo);
	bP_Lo_Trig 		 	:= xGR_MINR_P_Lo.Q AND bRelModul_ParaSetupOk;

	(* Operation mode selector switch *)
	bOMSS_MAT := (IN_EG.iIdx_OMSS = 1) OR (IN_EG.iIdx_OMSS = 2) OR (IN_EG.iIdx_OMSS = 3);	(* 1= manual; 2= auto; 3= test mode *)

	(* operation mode *)
	xOpMode.in	:=	IN_EG.iSt_OpMode;
	xOpMode();

END_PROGRAM
```

#### GeneralEG.var - Local variables
```iecst
VAR
	xGR_MAXR_StartSpd : GR_MAXR := (0); (*Engine start speed passed*)
	xGR_MINR_P_Lo : GR_MINR := (0); (*FuB*)
	xTOF_StartSpd : TOF := (0); (*FuB*)
	xTON_ParaSetupOk : TON := (0); (*FuB*)
END_VAR
```

### Program Logical/EngineGeneral/DefaultEG (IEC, version 4.14.0) - Settings default values

#### DefaultEGCyclic.st - Cyclic code
```iecst
(*******************************************************************************
DefaultEG		value set

This code is confidential and proprietary to the INNIO Company.
It may not be used in any form, or reproduced in any manner,
without the express written permission of the INNIO Company.
Copyright, INNIO Company, 2025

Customized modifications: -
------------------------

History:
-------
V03.99.00.00	18.03.2013	Tinello		new
V04.02.00		28.07.2015 	Plattner 	new
V4.14.0 		11.04.2025	Tinello		SAFETY related:	tSafetyLoop_EmStop added to get rid of problems during simulation

Instructions for use:
--------------------
- Default TRUE setting for not existing Di's

Outstandings:
------------

*******************************************************************************)

PROGRAM _CYCLIC

	(* default TRUE setting for not existing Di's *)
	IN_EG.tSafetyLoop_EmStop.Di 	:= IN_EG.tSafetyLoop_EmStop.Di 		OR NOT IN_EG.tSafetyLoop_EmStop.GoodQual; 	(* SAFETY PLC *)
	IN_EG.tSafetyLoop_Eng.Di 		:= IN_EG.tSafetyLoop_Eng.Di 		OR NOT IN_EG.tSafetyLoop_Eng.GoodQual;	(* old: RUHE *)
	IN_EG.tEmStop_CoolRun.Di 		:= IN_EG.tEmStop_CoolRun.Di  		OR NOT IN_EG.tEmStop_CoolRun.GoodQual;	(* emergency stop with cool down run *)

END_PROGRAM
```

### Program Logical/EngineGeneral/slowdownT (IEC, version 4.09.0) - + slow down time

- slowdownTCyclic.st (not readable text: treated as protected, skipped)

- slowdownTInit.st (not readable text: treated as protected, skipped)

#### slowdownT.var - Local variables
```iecst
VAR
	bCreateDataObj : BOOL; (*TRUE=create new data object *)
	bIgnoreMeasurement : BOOL := FALSE; (*Ignore measurement if speed gradient is not plausible for a certain time *)
	bIgnoreMeasuring : BOOL := FALSE; (*Ignore measuring if speed gradient not plausible*)
	bRel_Measuring : BOOL := FALSE; (*Release measuring*)
	bResetSDT : BOOL; (*reset array of measurements*)
	bSpeed_15 : BOOL; (*15% of nominal speed reached*)
	bSpeed_95 : BOOL; (*95% of nominal speed reached*)
	bStartMeasuring : BOOL := FALSE; (*measuring active *)
	bWriteDataObj : BOOL; (*TRUE=write data object module *)
	DatObjCreate_01 : DatObjCreate; (*data object create *)
	DatObjDelete_PermMem : DatObjDelete; (*data object delete *)
	DatObjInfo_01 : DatObjInfo; (*data object info *)
	DatObjRead_01 : DatObjRead; (*data object read *)
	DatObjWrite_01 : DatObjWrite; (*data object write *)
END_VAR
VAR CONSTANT
	ERR_NOERROR : UINT := 0;
END_VAR
VAR
	i : INT := 0; (*counter*)
	iSDT_Cnt : INT := 0; (*counter for aligned slow down time*)
	ModulName : STRING[25]; (*module name of object*)
	perm_slowdown_vers : UINT; (*version*)
	pm_Error : UINT; (*permanent value error*)
	pm_id : UDINT; (*permanent value identifier*)
	pm_len : UDINT; (*permanent value lenght*)
	pm_p : UDINT; (*permanent value pointer*)
	pm_sdt : ParaSDT_typ; (*permanent memory tags*)
	rN_EngAct_Old : REAL := 0.0; (*Save actual engine speed for one cylce (100ms)*)
	rN_EngAct_Save : REAL := 0.0; (*Save actual engine speed*)
	rSDT_Avg : REAL := 0.0; (*average aligned slow down time*)
	rSDT_ECWT_Factor : REAL := 0.0; (*alignment factor by cooling water temperature*)
	rSDT_EOT_Factor : REAL := 0.0; (*alignment factor by engine oil temperature*)
	rSDT_N_Factor : REAL := 0.0; (*alignment factor by engine speed*)
	rSDT_Sum : REAL := 0.0; (*sum of aligned slow down time*)
	rSlowDownTime : REAL := 0.0; (*measured engine slow down time from 95% speed to 5% speed [s]*)
	rSpeedGradientTime : REAL; (*Time for calculating the speed gradient*)
	rT_ECW_Sum : REAL := 0.0; (*sum engine cooling water temperature [°C]*)
	rT_EO_Sum : REAL := 0.0; (*sum engine oil temperature [°C]*)
	rU_Exc_Sum : REAL := 0.0; (*sum excitation voltage [V]*)
	TON_WarnDelay : TON := (0); (*FuB*)
	TON_WritePMEM : TON := (0); (*delay write permanent memory*)
	tRealTime : rtctime_typ;
	ucIndexSDT : USINT; (*index for circular buffer*)
	ulChecksum : UDINT; (*parameter checksum value*)
	ulChecksumOld : UDINT; (*last vlaue of parameter checksum*)
	ulChkValue : UDINT; (*actual value of parameter pointer*)
	ulPMPointer : UDINT; (*adress of actual checksum value*)
	write_once : BOOL; (*write permanent memory once*)
	xDTGetTime_RPS : DTGetTime;
	xF_TRIG_M_GASV : F_TRIG; (*FuB*)
	xF_TRIG_Speed15 : F_TRIG; (*trigger for speed falls below 15% nominal speed*)
	xF_TRIG_Speed95 : F_TRIG; (*trigger for speed falls below 95% nominal speed*)
	xLCRLimScal : LCRLimScal; (*linear interpolation function for correction factors*)
	xTON_IgnoreMeasuring : TON; (*ignore measurement speed gradient not plausible*)
	TON_BlockMinFileAge : TON; (*waiting time without file write after successful performed write*)
	bBlock_MinFileAge : BOOL := FALSE; (*pause the perm file write after each sucessful write*)
	iPM_WriteCnt : UDINT; (* *) (*old VarName: usPMWriteCnt*)
END_VAR
```

### Program Logical/EngineGeneral/barometric (IEC, version 4.10.0) - barometric pressure

#### barometricCyclic.st - Zyklischer Code
```iecst
(*******************************************************************************
barometric		barometric pressure  					(CYCLIC)

This code is confidential AND proprietary to the INNIO Company.
It may NOT be used in any form, or reproduced in any manner,
without the express written permission of the INNIO Company.
Copyright, INNIO Company, 2021

Customized modifications: -
------------------------

History:
-------
V04.02.00.00	28.01.2015  Tinello		NEW specification
V04.04.00.00	22.06.2015	Tinello		Limitierung eingefügt
				20.10.2016	Tinello		Limitierung angepasst -> Spezi (c)
V04.05.00.00	22.01.2018	Tinello		Out-Schnittstelle für Ms-Störung hinzu
V04.10.00.00	28.01.2021	Tinello  	BugFix: Timer & other FuB's

Instructions FOR use:
--------------------
*******************************************************************************)
PROGRAM _CYCLIC

	(*--------------------------------------------------------------*)
	(* RESET of alarms and warnings and pre-settings				*)
	(*--------------------------------------------------------------*)
	bAMM_Pr_Baro_Ms				:= FALSE;
	bAMM_Pr_Baro_siteDev_Lo		:= FALSE;
	bAMM_Pr_Baro_siteDev_Hi		:= FALSE;

	OUT_EG.rPr_Baro_Internal	:= 0;

	(*--------------------------------------------------------------*)
	(* VISU var of module 											*)
	(*--------------------------------------------------------------*)
	MM2VIS.rPr_Baro				:= IN_EG.tPr_Baro.Ai;

	(************************************************************************************************************************************)
	(************************              				  error monitoring		 	             	           **************************)
	(************************************************************************************************************************************)
	xGR_MINR_Baro(In:= IN_EG.tPr_Baro.Ai, Gw:= (Para.rPr_Baro_site - Para.rPr_Baro_siteDevMax), Hy:= 0.01); (* hyst. = 10 mbar *)
	xGR_MAXR_Baro(In:= IN_EG.tPr_Baro.Ai, Gw:= (Para.rPr_Baro_site + Para.rPr_Baro_siteDevMax), Hy:= 0.01);	(* hyst. = 10 mbar *)

	IF bRelModul_ParaSetupOk THEN

		(*----------------------------------------------------------*)
		(* measurement signal failure 								*)
		(*----------------------------------------------------------*)
		bAMM_Pr_Baro_Ms	 		:= Para.bPr_Baro_Exist 	AND NOT IN_EG.tPr_Baro.GoodQual;										(* W3449 *)

			(* Release monitoring *)
			xTOF_AMM_Pr_Baro(IN := bAMM_Pr_Baro_Ms, PT:= T#10s);					(* TOF because of filtered signals *)

			bRelMon_Pr_Baro		:= Para.bPr_Baro_Exist  AND NOT xTOF_AMM_Pr_Baro.Q;

		(*----------------------------------------------------------*)
		(* barometric pressure										*)
		(*----------------------------------------------------------*)
		bAMM_Pr_Baro_siteDev_Lo	:= xGR_MINR_Baro.Q AND bRelMon_Pr_Baro;															(* W2552 *)
		bAMM_Pr_Baro_siteDev_Hi	:= xGR_MAXR_Baro.Q AND bRelMon_Pr_Baro;															(* W2553 *)

		(* switch barometric pressure in case of error *)
		IF 	NOT bRelMon_Pr_Baro 	OR												(* sensor not active or measuring signal error *)
			bAMM_Pr_Baro_siteDev_Lo OR 												(* signal out of plausible range *)
			bAMM_Pr_Baro_siteDev_Hi
		THEN
			xRAMPE_R_Pr_Baro.In	:= Para.rPr_Baro_site;								(* use parameter for calculation *)
		ELSE
			xRAMPE_R_Pr_Baro.In	:= IN_EG.tPr_Baro.Ai;
		END_IF

		xRAMPE_R_Pr_Baro(enable	:= TRUE);

		OUT_EG.rPr_Baro_Internal		:= LIMIT(0.8, xRAMPE_R_Pr_Baro.Out, 1.050);	(* ramp with 10 mbar/s *)
		OUT_EG.bAMM_Pr_Baro_Internal	:= NOT bRelMon_Pr_Baro;
	ELSE
		xTOF_AMM_Pr_Baro(IN 			:= FALSE);
		xRAMPE_R_Pr_Baro(enable			:= FALSE);
	END_IF

END_PROGRAM
```

#### barometricInit.st
```iecst
(*******************************************************************************
barometric		barometric pressure  					(INIT)

This code is confidential AND proprietary to the INNIO Company.
It may NOT be used in any form, or reproduced in any manner,
without the express written permission of the INNIO Company.
Copyright, INNIO Company, 2019

Customized modifications: -
------------------------

History:
-------
V04.02.00.00	  28.01.2015  Tinello	NEW specification

Instructions FOR use:
--------------------
*******************************************************************************)
PROGRAM _INIT

	(* ramp settings *)
	xRAMPE_R_Pr_Baro.enable		:= TRUE;
	xRAMPE_R_Pr_Baro.Rise		:= 0.010;		(* 10 mbar/s *)
	xRAMPE_R_Pr_Baro.Sink		:= 0.010;		(* 10 mbar/s *)
	xRAMPE_R_Pr_Baro.TC_Time	:= TASK_TIME_100MS;

END_PROGRAM
```

#### barometric.var - Lokale Variablen
```iecst
VAR
	bRelMon_Pr_Baro : BOOL := FALSE; (*Release monitoring barometric pressure*)
END_VAR
VAR CONSTANT
	TASK_TIME_100MS : UINT := 100; (*Taskklassen Zeit 100ms *)
END_VAR
VAR
	xGR_MAXR_Baro : GR_MAXR := (0); (*FuB*)
	xGR_MINR_Baro : GR_MINR := (0); (*FuB*)
	xRAMPE_R_Pr_Baro : RAMPE_R := (0); (*FuB*)
	xTOF_AMM_Pr_Baro : TOF := (0); (*FuB*)
END_VAR
```

### Program Logical/EngineGeneral/MainBearing (IEC, version 4.05.3) - Main bearing temperature monitoring

#### MainBearingCyclic.st - Cyclic code
```iecst
(*******************************************************************************
MainBearing: main bearing temperature monitoring (cyclic)

This code is confidential and proprietary to the INNIO Company.
It may not be used in any form, or reproduced in any manner, without the express
written permission of the INNIO Company.
Copyright, INNIO Company, 2019

- reading main bearing temperature values
- sensor check
- warning main bearing temperature maximum monitoring
- error main bearing temperature maximum monitoring

Customized modifications: -
------------------------

History:
-------
V3.2		17-03-2010	Tinello, 	generated
V3.20.1		09-03-2011	Zengerer	eleminate temp to 0 in case of signal failure
			10-03-2011	Tinello		MS-Sto set to 140°C
V3.3		27.03.2013	Tinello 	restructured for modular SW
									add median monitoring
V3.59		14.01.2015	Tinello		restructured for XT4
V4.3		20.01.2016	Tinello		MIN, MAX AND AVG FOR temperature AND strength signal
V4.4		06.10.2016	Tinello		message "main bearing temperature MEDIAN deviation maximum" (with bearing position) added
V4.05.01.00	08.03.2018	Tinello		Specification (f)
V4.05.03.00	12.09.2018	Tinello		Bugfix: Alarm bypass, bu

Instructions for use:
--------------------

Outstandings:
------------

*******************************************************************************)
PROGRAM _CYCLIC

	(*--------------------------------------------------*)
	(* RESET 						 					*)
	(*--------------------------------------------------*)
	xMEDIAN_Temp.anzahl	:= 0;

	rT_MBearing_Min		:= 10000;
	rT_MBearing_Max		:= 0;
	rT_MBearing_Sum		:= 0;

	(************************************************************************************************************************)
	(************************              Monitoring of main bearing temperature		           **************************)
	(************************************************************************************************************************)
	FOR iCntMB := 1 TO 11 BY 1 DO																	(* 11 main bearings *)

		rT_MBearing[iCntMB]			:= IN_EG.tT_MBearing[iCntMB].Ai;

		(* error monitoring	*)
			(* TOF because of filtered signals *)
			xTOF_MBTempMs[iCntMB](IN:= NOT IN_EG.tT_MBearing[iCntMB].GoodQual, PT:= T#10s);

		bErrMBTemp_Ms[iCntMB] 		:= Para.bT_MBearing_Exist AND xTOF_MBTempMs[iCntMB].Q;			(* Ms error *)

		bErrMBTemp_Hi[iCntMB] 		:= (rT_MBearing[iCntMB] > Para.rT_MBearing_Hi) 	 AND 			(* Maximum warning *)
									   Para.bT_MBearing_Exist AND IN_EG.tT_MBearing[iCntMB].GoodQual;

		bErrMBTemp_HiHi[iCntMB] 	:= (rT_MBearing[iCntMB] > Para.rT_MBearing_HiHi) AND 			(* Maximum error *)
									   Para.bT_MBearing_Exist AND IN_EG.tT_MBearing[iCntMB].GoodQual;

		IF NOT bErrMBTemp_Ms[iCntMB] THEN
			xMEDIAN_Temp.anzahl						:= xMEDIAN_Temp.anzahl + 1;
			xMEDIAN_Temp.in[xMEDIAN_Temp.anzahl]	:= rT_MBearing[iCntMB];							(* median calculation *)
		END_IF

		bErrMBTempMDev_Lo[iCntMB]	:= (rT_MBearing[iCntMB] < (xMEDIAN_Temp.median - 				(* Negative deviation *)
										 						Para.rT_MBearing_MDev_HiHi)) AND
									    Para.bT_MBearing_Exist AND NOT bErrMBTemp_Ms[iCntMB];

		bErrMBTempMDev_HiHi[iCntMB]	:= (rT_MBearing[iCntMB] > (xMEDIAN_Temp.median + 				(* Positive deviation *)
										 						Para.rT_MBearing_MDev_HiHi)) AND
									    Para.bT_MBearing_Exist AND NOT bErrMBTemp_Ms[iCntMB];
	END_FOR

	(* Create MEDIAN *)
	xMEDIAN_Temp();

	(************************************************************************************************************************)
	(************************              			 AMM sequencer	 	             	           **************************)
	(************************************************************************************************************************)
	xTON_SecondTick(IN	:= NOT xTON_SecondTick.Q, PT:= T#800ms);							(* 800ms + 2x cycle time = 1 sec.*)
	xTON_ReleaseMDev(IN	:= IN_EG.rN_EngAct > 400, PT:= T#60s);								(* monitoring delay *)

	(* ERROR   main bearing temperature measuring signal failure  *)
	xAmmSeq_TempMs.Enable			:= NOT IN_EG.tAB2EG.bResetTrip AND bRelModul_ParaSetupOk;
	xAmmSeq_TempMs.ClockPulse		:= xTON_SecondTick.Q;
	xAmmSeq_TempMs.NrOfBits			:= 12;
	xAmmSeq_TempMs.BitArray			:= ADR(bErrMBTemp_Ms);
	xAmmSeq_TempMs();

	bAMM_T_MBearing_Ms				:= xAmmSeq_TempMs.Alarm1;														(* W9217 *)
	bOpM_T_MBearing_Ms				:= xAmmSeq_TempMs.Alarm2;														(* B2804 *)
	iNum_T_MBearing_Ms				:= xAmmSeq_TempMs.ErrorNr;

	(* WARNING main bearing temperature maximum  *)
	xAmmSeq_TempHi.Enable			:= NOT IN_EG.tAB2EG.bResetWarning;
	xAmmSeq_TempHi.ClockPulse		:= xTON_SecondTick.Q;
	xAmmSeq_TempHi.NrOfBits			:= 12;
	xAmmSeq_TempHi.BitArray			:= ADR(bErrMBTemp_Hi);
	xAmmSeq_TempHi();

	bAMM_T_MBearing_Hi				:= xAmmSeq_TempHi.Alarm1;														(* W2542 *)
	bOpM_T_MBearing_Hi				:= xAmmSeq_TempHi.Alarm2;														(* B2805 *)
	iNum_T_MBearing_Hi				:= xAmmSeq_TempHi.ErrorNr;

	(* ERROR   main bearing temperature maximum  *)
	xAmmSeq_TempHiHi.Enable			:= NOT IN_EG.tAB2EG.bResetTrip;
	xAmmSeq_TempHiHi.ClockPulse		:= xTON_SecondTick.Q;
	xAmmSeq_TempHiHi.NrOfBits		:= 12;
	xAmmSeq_TempHiHi.BitArray		:= ADR(bErrMBTemp_HiHi);
	xAmmSeq_TempHiHi();

	bAMM_T_MBearing_HiHi			:= xAmmSeq_TempHiHi.Alarm1;														(* A2228 *)

	(* WARNING   main bearing temperature - negative MEDIAN deviation maximum  *)
	xAmmSeq_TempMDevLo.Enable		:= NOT IN_EG.tAB2EG.bResetWarning AND xTON_ReleaseMDev.Q;
	xAmmSeq_TempMDevLo.ClockPulse	:= xTON_SecondTick.Q;
	xAmmSeq_TempMDevLo.NrOfBits		:= 12;
	xAmmSeq_TempMDevLo.BitArray		:= ADR(bErrMBTempMDev_Lo);
	xAmmSeq_TempMDevLo();

	bAMM_T_MBearing_MDev_Lo			:= xAmmSeq_TempMDevLo.Alarm1;													(* W9218 *)
	bOpM_T_MBearing_MDev_Lo			:= xAmmSeq_TempMDevLo.Alarm2;													(* B2958 *)
	iNum_T_MBearing_MDev_Lo			:= xAmmSeq_TempMDevLo.ErrorNr;

	(* ERROR   main bearing temperature - positive MEDIAN deviation maximum  *)
	xAmmSeq_TempMDevHiHi.Enable		:= NOT (IN_EG.tAB2EG.bResetTrip OR (IN_EG.tAB2EG.bResetWarning AND bMsg2285_Test)) AND
									   xTON_ReleaseMDev.Q;
	xAmmSeq_TempMDevHiHi.ClockPulse	:= xTON_SecondTick.Q;
	xAmmSeq_TempMDevHiHi.NrOfBits	:= 12;
	xAmmSeq_TempMDevHiHi.BitArray	:= ADR(bErrMBTempMDev_HiHi);
	xAmmSeq_TempMDevHiHi();

	bAMM_T_MBearing_MDev_HiHi		:= xAmmSeq_TempMDevHiHi.Alarm1;													(* A2285 *)
	bOpM_T_MBearing_MDev_HiHi		:= xAmmSeq_TempMDevHiHi.Alarm2;													(* B2904 *)
	iNum_T_MBearing_MDev_HiHi		:= xAmmSeq_TempMDevHiHi.ErrorNr;

	(************************************************************************************************************************)
	(************************              					VISU	 	             	           **************************)
	(************************************************************************************************************************)
	FOR iCntMB := 1 TO 11 BY 1 DO
		MM2VIS.rT_MBearing[iCntMB]	:= rT_MBearing[iCntMB];
		OUT_EG.rT_MBearing[iCntMB]	:= rT_MBearing[iCntMB];			(* OUT interface - For other modules *)

		(* search for the bearing temperature - MIN,MAX,AVG *)
		rT_MBearing_Min				:= MIN(rT_MBearing_Min, rT_MBearing[iCntMB]);
		rT_MBearing_Max 			:= MAX(rT_MBearing_Max, rT_MBearing[iCntMB]);
		rT_MBearing_Sum				:= rT_MBearing_Sum + rT_MBearing[iCntMB];
	END_FOR

	MM2VIS.rT_MBearing_Min			:= rT_MBearing_Min;
	MM2VIS.rT_MBearing_Max			:= rT_MBearing_Max;
	MM2VIS.rT_MBearing_Avg			:= rT_MBearing_Sum / 11;

	MM2VIS.iNum_T_MBearing_MsMs		:= iNum_T_MBearing_Ms;
	MM2VIS.iNum_T_MBearing_Hi		:= iNum_T_MBearing_Hi;
	MM2VIS.iNum_T_MBearing_MDev_Lo	:= iNum_T_MBearing_MDev_Lo;
	MM2VIS.iNum_T_MBearing_MDev_HiHi:= iNum_T_MBearing_MDev_HiHi;

END_PROGRAM
```

#### MainBearing.var - Local variables
```iecst
VAR
	bErrMBTempMDev_HiHi : ARRAY[0..11] OF BOOL := [12(FALSE)]; (*main bearing temperature - positive deviation from Median - maximum error*)
	bErrMBTempMDev_Lo : ARRAY[0..11] OF BOOL := [12(FALSE)]; (*main bearing temperature - negative deviation from Median - maximum warning*)
	bErrMBTemp_Hi : ARRAY[0..11] OF BOOL := [12(FALSE)]; (*main bearing temperature - maximum warning*)
	bErrMBTemp_HiHi : ARRAY[0..11] OF BOOL := [12(FALSE)]; (*main bearing temperature - maximum error*)
	bErrMBTemp_Ms : ARRAY[0..11] OF BOOL := [12(FALSE)]; (*main bearing temperature - measurement signal failure *)
	iCntMB : USINT := 0; (*counter for main bearing number *)
	iNum_T_MBearing_Hi : USINT := 0; (*main bearing temperature maximum - bearing position (number)*)
	iNum_T_MBearing_MDev_HiHi : USINT := 0; (*main bearing temperature - positive deviation from MEDIAN maximum - bearing position (number)*)
	iNum_T_MBearing_MDev_Lo : USINT := 0; (*main bearing temperature - negative deviation from MEDIAN maximum - bearing position (number)*)
	iNum_T_MBearing_Ms : USINT := 0; (*main bearing temperature measurement signal failure - bearing position (number)*)
	rT_MBearing : ARRAY[0..11] OF REAL := [12(0.0)]; (*filtered main bearing temperature [°C]*)
	rT_MBearing_Max : REAL := 0.0; (*maximum main bearing temperature [°C]*)
	rT_MBearing_Min : REAL := 0.0; (*minimum main bearing temperature [°C]*)
	rT_MBearing_Sum : REAL := 0.0; (*sum of all main bearing temperature [°C]*)
	xAmmSeq_TempHi : AmmSequence := (0); (*FuB*)
	xAmmSeq_TempHiHi : AmmSequence := (0); (*FuB*)
	xAmmSeq_TempMDevHiHi : AmmSequence := (0); (*FuB*)
	xAmmSeq_TempMDevLo : AmmSequence := (0); (*FuB*)
	xAmmSeq_TempMs : AmmSequence := (0); (*FuB*)
	xMEDIAN_Temp : RMEDIAN24 := (0); (*FuB*)
	xTOF_MBTempMs : ARRAY[0..11] OF TOF := [12(0)]; (*FuB*)
	xTON_ReleaseMDev : TON := (0); (*FuB*)
	xTON_SecondTick : TON := (0); (*FuB*)
END_VAR
```

### Program Logical/EngineGeneral/ConRoMon (IEC, version 4.10.0) - conrod bearing temperature monitoring

#### ConRoMonCyclic.st - Cyclic code
```iecst
(*******************************************************************************
ConRoMon: Conrod bearing temperature CANopen Sensor (cyclic)

This code is confidential AND proprietary to the INNIO Company.
It may NOT be used in any form, or reproduced in any manner, without the express
written permission of the INNIO Company.
Copyright, INNIO Company, 2021

Customized modifications: -
------------------------

History:
-------
V0.1		27-05-2009	Kröll,Waldhart,Weigl generated
V0.11		22-03-2010	Waldhart,  	enhanced FOR 24 cylinder
V0.11.1		17-11-2010	Waldhart,  	only FOR BR9 active
V0.12		10-06-2011	Waldhart,  	alarms over-worked
			01-08-2011	Waldhart,  	alarms over-worked
V0.12.1		18-08-2011	Waldhart,  	over-worked
V0.13		27.03.2013	Tinello 	restructured FOR modular SW
									add median monitoring
V0.14		14.01.2015	Tinello	 	restructured FOR XT4
V4.3		20.01.2016	Tinello		calibration and parametrization; read signal strength;
									MIN, MAX and AVG for temperature and strength signal
V4.4		19.08.2016	Tinello		bugfix ACK A3378;
			06.09.2016	Tinello		CANQueue, LowLoad and fault tolerant mode added --> Specification (d)
									message "conrod bearing temperature MEDIAN deviation maximum" (with bearing position) added
V4.5		27.01.2017	Tinello		Specification (e)
			17.05.2017	Tinello		Specification (e) + release after 60s with 400rpm
V4.05.01.00	07.03.2018	Tinello		Specification (f)
V4.05.03.00	12.09.2018	Tinello		Bugfix: Alarm bypass, bu
V4.07.00.00	28.03.2019	Tinello		Bugfix: power was compared to 30 instead of 0.3
V4.10.00.00	28.01.2021	Tinello  	BugFix: Timer & other FuB's

Instructions FOR use:
--------------------

Outstandings:
------------

*******************************************************************************)
PROGRAM _CYCLIC

	(*--------------------------------------------------*)
	(* RESET of alarms and values	 					*)
	(*--------------------------------------------------*)
	bOpM_T_CBearing_Calib_Ok		:= FALSE;
	bWrongCylinder	 				:= FALSE;									(* reset wrong cylinder information bit *)

	rT_CBearing_Min					:= 10000;									(* reset min, max & avg temperature *)
	rT_CBearing_Max					:= 0;
	rT_CBearing_Sum					:= 0;

	iPc_T_CBearing_Sig_Min			:= 10000;									(* reset min, max & avg signal strength *)
	iPc_T_CBearing_Sig_Max			:= 0;
	iPc_T_CBearing_Sig_Sum			:= 0;

	iPc_T_CBearing_Gain_Min			:= 10000;									(* reset min, max & avg receiver gain level *)
	iPc_T_CBearing_Gain_Max			:= 0;
	iPc_T_CBearing_Gain_Sum			:= 0;

	iCntCB_MsOk						:= 0;										(* number of bearings with NO measurement error *)

	VIS2MM.iNum_T_CBearing_Calib	:= LIMIT(0, VIS2MM.iNum_T_CBearing_Calib, 20);

	(********************************************************************************************************************************)
	(************************             					 CAN communication				     	       **************************)
	(********************************************************************************************************************************)
	bRel_CBearing_CAN	:= Para.bT_CBearing_Exist	AND
						   NOT bAMM_T_CBearing_CAN	AND 						(* CAN bus communication - error *)
						   bRelModul_ParaSetupOk;

	(*--------------------------------------------------------------------------*)
	(* parametrization of kongsberg system per SDO's							*)
	(*--------------------------------------------------------------------------*)
	IF bAMM_T_CBearing_CAN THEN	 												(* send parameters again if CAN error *)
		iCnt_Para		:= 0;
		iSt_Para		:= 0;
		iCntCB_Para		:= 1;
	END_IF

	IF 	bRel_CBearing_CAN	AND													(* CAN bus released for read and write *)
		(iCnt_Para < 6) 			 											(* not all parameters have been transfered *)
	THEN
		(* load parameter settings *)
		CASE iCnt_Para OF
 			0:	(* Number of channels *)
				DATA_W.Address	:= 16#23;										(* 23 = WRITE with 4 databytes *)
				DATA_W.IndexHi	:= 16#21;
 				DATA_W.IndexLo	:= 16#02;
 				DATA_W.Data		:= 20;											(* 20 channels *)

  			1:	(* Minimum expected engine speed *)
				DATA_W.Address	:= 16#23;
				DATA_W.IndexHi	:= 16#21;
 				DATA_W.IndexLo	:= 16#01;
 				DATA_W.Data		:= 400;											(* 400 rpm *)

  			2:	(* Temperature value wenn sensor not detected *)
				DATA_W.Address	:= 16#23;
				DATA_W.IndexHi	:= 16#21;
 				DATA_W.IndexLo	:= 16#12;
 				DATA_W.Data		:= 1;											(* Temp = 0 if engine is not running *)

  			3:	(* High temperature alarm limit *)
				DATA_W.Address	:= 16#23;
				DATA_W.IndexHi	:= 16#20;
 				DATA_W.IndexLo	:= 16#09;
 				DATA_W.Data		:= 125;											(* 125 °C *)

			4:	(* HighHigh temperature alarm limit *)
				DATA_W.Address	:= 16#23;
				DATA_W.IndexHi	:= 16#20;
 				DATA_W.IndexLo	:= 16#0A;
 				DATA_W.Data		:= 130;											(* 130 °C *)

			5:	(* Delay before alarm output is set *)
				DATA_W.Address	:= 16#23;
				DATA_W.IndexHi	:= 16#20;
 				DATA_W.IndexLo	:= 16#0B;
 				DATA_W.Data		:= 0;											(* 0 sec. *)
		END_CASE

		(* prepare writing of parameters *)
		CASE iSt_Para OF
			0:	iSt_Para		:= 1;

			1:	(* write parameter *)
				xTON_WriteMax(IN:= FALSE);
				xTON_WriteAck(IN:= FALSE);
				iSt_Para		:= 2;

			2:	(* check parameter set *)
				IF iCnt_Para > 2 THEN
					xTON_WriteMax.PT	:= T#500ms;
					xTON_WriteAck.PT	:= T#300ms;
				ELSE
					xTON_WriteMax.PT 	:= T#6s;
					xTON_WriteAck.PT	:= T#5s;
				END_IF

				xTON_WriteMax(IN:= TRUE);										(* max time to acknowledge parameter set *)
				xTON_WriteAck(IN:= (DATA_R.Address  = 16#60) 	 		AND		(* timer to detect writing errors *)
							 	   (DATA_R.IndexHi  = DATA_W.IndexHi)	AND
								   (DATA_R.IndexLo  = DATA_W.IndexLo)	AND
								   (DATA_R.Cylinder = DATA_W.Cylinder)		);

				IF xTON_WriteAck.Q THEN

					(* parameter set was OK *)
					iSt_Para		:= 0;

					IF  (iCntCB_Para < xEngType.NumberOfCylinder) AND
						(iCnt_Para 	 > 2)
					THEN
						iCntCB_Para	:= iCntCB_Para + 1;
					ELSE
						iCnt_Para 	:= iCnt_Para + 1;
						iCntCB_Para	:= 1;
					END_IF

				ELSIF xTON_WriteMax.Q THEN
					iSt_Para		:= 1;										(* write parameter again *)
				END_IF
		END_CASE

		IF iCnt_Para > 2 THEN	DATA_W.Cylinder	:= iCntCB_Para;
						 ELSE	DATA_W.Cylinder	:= 0;							(* only one parameter for all cylinders *)
		END_IF
	ELSE
		xTON_WriteMax(IN:= FALSE);
		xTON_WriteAck(IN:= FALSE);
	END_IF

	(*--------------------------------------------------------------------------*)
	(* calibration of kongsberg system per SDO's								*)
	(*--------------------------------------------------------------------------*)
	IF	NOT bRel_CBearing_CAN								OR					(* CAN bus NOT released for read and write *)
		(iCnt_Para < 6) 		 							OR	  				(* parameter set NOT finished *)
		(iSt_ReadStrength > 0)								OR					(* reading of signal strength active *)
		MM2VIS.bMsg2794										OR					(* conrod bearing temp. calibration unsuccessful *)
		((IN_EG.rN_EngAct < 400) AND (iNumCB_Calib = 0))  	OR					(* calibration of all cyl. only during engine run *)
 		NOT VIS2MM.bDem_T_CBearing_Calib
	THEN
		VIS2MM.bDem_T_CBearing_Calib	:= FALSE;								(* reset demand *)

		iNumCB_Calib 			:= INT_TO_USINT(VIS2MM.iNum_T_CBearing_Calib);	(* bearing position not changeable during calibr. *)
		iSt_Calib				:= 0;
		iCntCB_Calib			:= 1;
	ELSE
		CASE iSt_Calib OF
			(* write calibration demand *)
			0:	DATA_W.Address	:= 16#23; 										(* 23 = WRITE with 4 databytes *)
				DATA_W.IndexHi	:= 16#20;										(* index 2021 = calibration of cable delay *)
				DATA_W.IndexLo	:= 16#21;
				DATA_W.Data		:= 1;											(* 1: start calibration *)
				iSt_Calib		:= 1;

			1:	IF (iCntCB_Calib < xEngType.NumberOfCylinder) AND
				   (iNumCB_Calib = 0) 											(* 0 = calibrate all cylinders *)
				THEN
					iCntCB_Calib	:= iCntCB_Calib + 1;
				ELSE
					iCntCB_Calib	:= 1;
					iSt_Calib		:= 2;
				END_IF

			(* write read command: state of calibration *)
			2:	DATA_W.Address	:= 16#40; 										(* 40 = READ *)
				DATA_W.IndexHi	:= 16#20;										(* index 2002 = state *)
				DATA_W.IndexLo	:= 16#02;
				DATA_W.Data		:= 0;
				iSt_Calib		:= 3;

			3:	iSt_Calib		:= 4;

			(* read state of calibration *)
			4:	IF 	(DATA_R.Address  = 16#4F) 		AND
					(DATA_R.IndexHi  = 16#20) 		AND
					(DATA_R.IndexLo  = 16#02) 		AND
					(DATA_R.Cylinder = DATA_W.Cylinder)
				THEN
					MM2VIS.iSt_T_CBearing_Calib[DATA_R.Cylinder]	:= DATA_R.Data + 1;
					iSt_Calib		:= 3;

					IF (iCntCB_Calib < xEngType.NumberOfCylinder) AND
					   (iNumCB_Calib = 0) 										(* 0 = read status of all cylinders *)
					THEN
						iCntCB_Calib	:= iCntCB_Calib + 1;
					ELSE
						iCntCB_Calib	:= 1;
					END_IF
				END_IF

				IF xTON_Calibration.Q THEN  iSt_Calib	:= 5; END_IF

			(* check state of calibration after 120s *)
			5:	FOR i:= 1 TO xEngType.NumberOfCylinder DO
   					IF (MM2VIS.iSt_T_CBearing_Calib[i] = 4) OR
					   ((iNumCB_Calib <> i) AND (iNumCB_Calib <> 0))

					THEN 	bCalib_Again[i]	:= FALSE;
		  		  	ELSE	bCalib_Again[i]	:= TRUE;
							iSt_Calib		:= 6;
					END_IF
				END_FOR

				IF iSt_Calib = 5 THEN
					VIS2MM.bDem_T_CBearing_Calib	:= FALSE; 					(* Calibration DONE - reset demand *)
					bReadStrength					:= TRUE;					(* Read signal strength after calibration *)
					bOpM_T_CBearing_Calib_Ok		:= TRUE;																(* B2909 *)
				END_IF

			(* write calibration demand AGAIN *)
			6:	DATA_W.Address	:= 16#23; 										(* 23 = WRITE with 4 databytes *)
				DATA_W.IndexHi	:= 16#20;										(* index 2021 = calibration of cable delay *)
				DATA_W.IndexLo	:= 16#21;
				DATA_W.Data		:= 1;											(* 1: start calibration *)

				iNumCalib_Again	:= 0;

				FOR i:= 1 TO xEngType.NumberOfCylinder DO
					IF	bCalib_Again[i] AND iNumCalib_Again = 0 THEN
						iNumCalib_Again	:= i;
						bCalib_Again[i]	:= FALSE;
					END_IF
				END_FOR

				IF iNumCalib_Again = 0 THEN iSt_Calib	:= 2; END_IF
		END_CASE

		IF iSt_Calib = 6			THEN	DATA_W.Cylinder	:= iNumCalib_Again;
		ELSIF (iNumCB_Calib = 0) 	THEN	DATA_W.Cylinder	:= iCntCB_Calib;
									ELSE	DATA_W.Cylinder	:= iNumCB_Calib;
		END_IF
	END_IF

	xTON_Calibration(IN		:= iSt_Calib > 1, PT:= T#180s);
	bAMM_T_CBearing_Calib	:= Para.bT_CBearing_Exist AND xTON_Calibration.Q;												(* W2794 *)

	(*--------------------------------------------------------------------------*)
	(* read signal strength and signal gain factor per SDO's					*)
	(*--------------------------------------------------------------------------*)
	xTON_ReadStrength(IN:= IN_EG.rN_EngAct >= Para.rN_EngNom * 0.95, PT:= T#2h);

	IF 	xTON_ReadStrength.Q															OR		(* read - every 2h *)
		EDGEPOS( IN_EG.rN_EngAct >= Para.rN_EngNom * 0.95) 							OR 		(* read - at engine start *)
		EDGENEG((IN_EG.rN_EngAct >= Para.rN_EngNom * 0.95) AND IN_EG.bEng_Aux_Dem)			(* read - at engine stop *)
	THEN
		bReadStrength		:= TRUE;
		xTON_ReadStrength(IN:= FALSE);
	END_IF

	IF EDGENEG(IN_EG.rN_EngAct > Para.rN_EngNom * 0.4) THEN  bReadStrength	:= FALSE;	END_IF

	IF	bRel_CBearing_CAN		AND												(* CAN bus released for read and write *)
		(iCnt_Para >= 6) 		AND	 											(* all parameters have been transfered *)
		(iSt_Calib =  0)		AND												(* calibration not active *)
	 	bReadStrength
	THEN
		CASE iSt_ReadStrength OF
			(* write read command: strength of the signal from the sensor *)
			0:	DATA_W.Address		:= 16#40; 									(* 40 = READ *)
				DATA_W.IndexHi		:= 16#20;									(* index 2006 = strength of signal *)
				DATA_W.IndexLo		:= 16#06;
				DATA_W.Data			:= 0;
				iSt_ReadStrength	:= 1;

			1:	iSt_ReadStrength	:= 2;

			(* read strength of signal *)
			2:	IF 	(DATA_R.Address  = 16#4F) 		AND
					(DATA_R.IndexHi  = 16#20) 		AND
					(DATA_R.IndexLo  = 16#06) 		AND
					(DATA_R.Cylinder = DATA_W.Cylinder)
				THEN
					iPc_T_CBearing_Sig_Act[DATA_R.Cylinder].Act[iCntCB_ReadAct]	:= DATA_R.Data;

					iSt_ReadStrength		:= 1;								(* write next read command *)

					IF (iCntCB_Read < xEngType.NumberOfCylinder)
					THEN
						iCntCB_Read			:= iCntCB_Read + 1;
					ELSE
						iCntCB_Read			:= 1;
						iCntCB_ReadAct		:= iCntCB_ReadAct + 1;

						IF iCntCB_ReadAct > 10 THEN

							FOR i:= 1 TO xEngType.NumberOfCylinder BY 1 DO

								iPc_T_CBearing_Sig_ActSum		:= 0;

								FOR ii:= 1 TO 10 DO
									iPc_T_CBearing_Sig_ActSum	:= iPc_T_CBearing_Sig_ActSum + iPc_T_CBearing_Sig_Act[i].Act[ii];
								END_FOR

								MM2VIS.iPc_T_CBearing_Sig[i]	:= iPc_T_CBearing_Sig_ActSum / 10;
							END_FOR

							iSt_ReadGain 		:= 1;							(* start reading the receiver gain level *)
							iCntCB_Read			:= 1;
							iCntCB_ReadAct		:= 1;

							iSt_ReadStrength	:= 3;							(* reading of signal strength done *)
						END_IF
					END_IF
				END_IF

			(* reading of signal strength done *)
			3:	iSt_ReadStrength	:= 3;
		END_CASE

		CASE iSt_ReadGain OF
			(* wait until reading of signal strength done *)
			0:	iSt_ReadGain		:= 0;

			(* write read command: receiver gain level *)
			1:	DATA_W.Address		:= 16#40; 									(* 40 = READ *)
				DATA_W.IndexHi		:= 16#20;									(* index 2005 = receiver gain level *)
				DATA_W.IndexLo		:= 16#05;
				DATA_W.Data			:= 0;
				iSt_ReadGain		:= 2;

			2:	iSt_ReadGain		:= 3;

			(* read receiver gain level *)
			3:	IF 	(DATA_R.Address  = 16#4F) 		AND
					(DATA_R.IndexHi  = 16#20) 		AND
					(DATA_R.IndexLo  = 16#05) 		AND
					(DATA_R.Cylinder = DATA_W.Cylinder)
				THEN
					iPc_T_CBearing_Gain_Act[DATA_R.Cylinder].Act[iCntCB_ReadAct]	:= DATA_R.Data;

					iSt_ReadGain			:= 2;								(* write next read command *)

					IF (iCntCB_Read < xEngType.NumberOfCylinder)
					THEN
						iCntCB_Read			:= iCntCB_Read + 1;
					ELSE
						iCntCB_Read			:= 1;
						iCntCB_ReadAct		:= iCntCB_ReadAct + 1;

						IF iCntCB_ReadAct > 10 THEN

							FOR i:= 1 TO xEngType.NumberOfCylinder BY 1 DO

								iPc_T_CBearing_Gain_ActSum		:= 0;

								FOR ii:= 1 TO 10 DO
									iPc_T_CBearing_Gain_ActSum	:= iPc_T_CBearing_Gain_ActSum + iPc_T_CBearing_Gain_Act[i].Act[ii];
								END_FOR

								MM2VIS.iPc_T_CBearing_Gain[i]	:= iPc_T_CBearing_Gain_ActSum / 10;
							END_FOR

							bReadStrength 	:= FALSE;
						END_IF
					END_IF
				END_IF
		END_CASE

		DATA_W.Cylinder		:= iCntCB_Read;
	ELSE
		(* reset *)
		iSt_ReadStrength	:= 0;
		iSt_ReadGain		:= 0;
		iCntCB_Read			:= 1;
		iCntCB_ReadAct		:= 1;
	END_IF

	(*--------------------------------------------------------------------------*)
	(* CAN BUS - WRITE & READ													*)
	(*--------------------------------------------------------------------------*)
	(* write demand to kongsberg system *)
	IF (iSt_Para  = 1) OR
	   (iSt_Calib = 1) OR (iSt_Calib = 3) OR (iSt_Calib = 6) OR
	   (iSt_ReadStrength = 1)								 OR
	   (iSt_ReadGain = 2)
	THEN
		xCANwrite_CB_Data.enable 	:= TRUE;
		xCANwrite_CB_Data.us_ident	:= IN_EG.iCAN_CB_us_ident;
		xCANwrite_CB_Data.can_id	:= 16#604;									(* set can identifier (600 plus Node-ID) *)
		xCANwrite_CB_Data.data_adr	:= ADR(DATA_W);
		xCANwrite_CB_Data.data_lng	:= 8;
		xCANwrite_CB_Data();
	END_IF

	(* read the acknowledge info *)
	IF (iSt_Para = 2) OR (iSt_Calib = 4) OR (iSt_ReadStrength = 2) OR (iSt_ReadGain = 3)
	THEN
		xCANread_CB_Data.enable 	:= TRUE;
		xCANread_CB_Data.us_ident	:= IN_EG.iCAN_CB_us_ident;
		xCANread_CB_Data.can_id		:= 16#584;									(* set can identifier (580 plus Node-ID) *)
		xCANread_CB_Data.data_adr	:= ADR(DATA_R);
		xCANread_CB_Data();
	END_IF

	(*--------------------------------------------------------------------------*)
	(* Read conrod bearing temperature via PDO's	 							*)
	(*--------------------------------------------------------------------------*)
	memset(ADR(TEMP), 0, SIZEOF(TEMP));											(* clear received data *)

	IF (IN_EG.iCAN_CB_us_ident <> 0) AND NOT bQueueInitDone THEN
		(* generate CANqueue *)
		xCANqueue_CB_Temp.enable	:= TRUE;
		xCANqueue_CB_Temp.us_ident	:= IN_EG.iCAN_CB_us_ident;					(* set us_ident with the value from CANopen *)
		xCANqueue_CB_Temp.can_id	:= 16#184;									(* set can identifier (180 plus Node-ID) *)
		xCANqueue_CB_Temp.size		:= 100;										(* number of telegrams in the queue *)
		xCANqueue_CB_Temp;

		IF xCANqueue_CB_Temp.status = 0 THEN
			bQueueInitDone	:= TRUE;
		END_IF
	END_IF

	IF xCANqueue_CB_Temp.us_ident <> 0 THEN
		(* read CANqueue *)
		xCANrd_CB_Temp.enable	:= TRUE;
		xCANrd_CB_Temp.q_ident	:= xCANqueue_CB_Temp.q_ident;					(* set q_ident with the value from CANqueue *)
		xCANrd_CB_Temp.data_adr	:= ADR(TEMP);									(* set data address *)
		xCANrd_CB_Temp();
	ELSE
		xCANrd_CB_Temp(enable	:= FALSE);
	END_IF

	CASE TEMP.Cylinder OF
		0: 																		(* wait for new data		*)
		1:	rT_CBearing[1]		:= UINT_TO_REAL(TEMP.Data);						(* temperature cylinder  1	*)
		2:	rT_CBearing[2]		:= UINT_TO_REAL(TEMP.Data);						(* temperature cylinder  2 	*)
		3:	rT_CBearing[3]		:= UINT_TO_REAL(TEMP.Data);						(* temperature cylinder  3 	*)
		4:	rT_CBearing[4]		:= UINT_TO_REAL(TEMP.Data);						(* temperature cylinder  4 	*)
		5:	rT_CBearing[5]		:= UINT_TO_REAL(TEMP.Data);						(* temperature cylinder  5 	*)
		6:	rT_CBearing[6]		:= UINT_TO_REAL(TEMP.Data);						(* temperature cylinder  6 	*)
		7:	rT_CBearing[7]		:= UINT_TO_REAL(TEMP.Data);						(* temperature cylinder  7 	*)
		8:	rT_CBearing[8]		:= UINT_TO_REAL(TEMP.Data);						(* temperature cylinder  8 	*)
		9:	rT_CBearing[9]		:= UINT_TO_REAL(TEMP.Data);						(* temperature cylinder  9 	*)
		10:	rT_CBearing[10]		:= UINT_TO_REAL(TEMP.Data);						(* temperature cylinder 10 	*)
		11:	rT_CBearing[11]		:= UINT_TO_REAL(TEMP.Data);						(* temperature cylinder 11 	*)
		12:	rT_CBearing[12]		:= UINT_TO_REAL(TEMP.Data);						(* temperature cylinder 12 	*)
		13:	rT_CBearing[13] 	:= UINT_TO_REAL(TEMP.Data);						(* temperature cylinder 13 	*)
		14:	rT_CBearing[14]		:= UINT_TO_REAL(TEMP.Data);						(* temperature cylinder 14 	*)
		15:	rT_CBearing[15]		:= UINT_TO_REAL(TEMP.Data);						(* temperature cylinder 15 	*)
		16:	rT_CBearing[16]		:= UINT_TO_REAL(TEMP.Data);						(* temperature cylinder 16 	*)
		17:	rT_CBearing[17]		:= UINT_TO_REAL(TEMP.Data);						(* temperature cylinder 17 	*)
		18:	rT_CBearing[18]		:= UINT_TO_REAL(TEMP.Data);						(* temperature cylinder 18 	*)
		19:	rT_CBearing[19]		:= UINT_TO_REAL(TEMP.Data);						(* temperature cylinder 19 	*)
		20:	rT_CBearing[20] 	:= UINT_TO_REAL(TEMP.Data);						(* temperature cylinder 20 	*)

		ELSE
			bWrongCylinder		:= bRelModul_ParaSetupOk;						(* wrong cylinder information *)
	END_CASE

	(*--------------------------------------------------*)
	(* Monitoring of CAN communication					*)
	(*--------------------------------------------------*)
	xTON_CANread(IN:= (xCANrd_CB_Temp.status <> 0) AND bRelModul_ParaSetupOk AND NOT IN_EG.tAB2EG.bResetWarning, PT:= T#10s);
	xTON_CANopen(IN:= (IN_EG.iCAN_CB_us_ident = 0) AND bRelModul_ParaSetupOk AND NOT IN_EG.tAB2EG.bResetWarning, PT:= T#10s);
	xTON_ParaSet(IN:= (iCnt_Para < 6) 			   AND bRelModul_ParaSetupOk AND NOT IN_EG.tAB2EG.bResetWarning, PT:= T#80s);

	bAMM_T_CBearing_CAN	:= Para.bT_CBearing_Exist  AND (xTON_CANopen.Q OR xTON_CANread.Q OR 								(* A2229 *)
												 	    xTON_ParaSet.Q OR bWrongCylinder);

	(********************************************************************************************************************************)
	(************************     	         Monitoring of conrod bearing temperature			           **************************)
	(********************************************************************************************************************************)
	FOR iCntCB:= 1 TO xEngType.NumberOfCylinder BY 1 DO

		(* actual temperature *)
		MM2VIS.rT_CBearing[iCntCB]			:= rT_CBearing[iCntCB];				(* visu *)
		OUT_EG.rT_CBearing[iCntCB]			:= rT_CBearing[iCntCB];				(* OUT interface - For other modules *)

		(* search for signal strength MIN, MAX, SUM --> AVG *)
		iPc_T_CBearing_Sig_Min				:= MIN(iPc_T_CBearing_Sig_Min,  MM2VIS.iPc_T_CBearing_Sig[iCntCB]);
		iPc_T_CBearing_Sig_Max				:= MAX(iPc_T_CBearing_Sig_Max,  MM2VIS.iPc_T_CBearing_Sig[iCntCB]);
		iPc_T_CBearing_Sig_Sum				:= iPc_T_CBearing_Sig_Sum   +   MM2VIS.iPc_T_CBearing_Sig[iCntCB];

		(* search for receiver gain level MIN, MAX, SUM --> AVG *)
		iPc_T_CBearing_Gain_Min				:= MIN(iPc_T_CBearing_Gain_Min, MM2VIS.iPc_T_CBearing_Gain[iCntCB]);
		iPc_T_CBearing_Gain_Max				:= MAX(iPc_T_CBearing_Gain_Max, MM2VIS.iPc_T_CBearing_Gain[iCntCB]);
		iPc_T_CBearing_Gain_Sum				:= iPc_T_CBearing_Gain_Sum   +  MM2VIS.iPc_T_CBearing_Gain[iCntCB];

		(* Only intact signals used for calculation *)
		IF rT_CBearing[iCntCB] > 5 THEN
			iCntCB_MsOk						:= iCntCB_MsOk + 1;					(* number of bearings without measurement error *)

			(* search for bearing temperature MIN, MAX, SUM --> AVG *)
			rT_CBearing_Min					:= MIN(rT_CBearing_Min, rT_CBearing[iCntCB]);
			rT_CBearing_Max					:= MAX(rT_CBearing_Max, rT_CBearing[iCntCB]);
			rT_CBearing_Sum					:= rT_CBearing_Sum   +  rT_CBearing[iCntCB];

			(* temperature median calculation *)
			xMEDIAN_Temp.in[iCntCB_MsOk]	:= rT_CBearing[iCntCB];
		END_IF
	END_FOR

	(* Create MEDIAN *)
	xMEDIAN_Temp.anzahl		:= iCntCB_MsOk;
	xMEDIAN_Temp();

	(* error monitoring *)
	xGR_MINR_T_EO(In:= IN_EG.tT_EO.Ai, Gw:= 65, Hy:= 5); 						(* hyst. = 5 °C *)
	xGR_MAXR_T_EO(In:= IN_EG.tT_EO.Ai, Gw:= 65, Hy:= 5);						(* hyst. = 5 °C *)

		IF EDGEPOS(xGR_MINR_T_EO.Q) OR EDGENEG(xGR_MAXR_T_EO.Q) THEN	bAdd_CBearing_Hi_Offset	:= FALSE; 	END_IF
		IF EDGENEG(xGR_MINR_T_EO.Q) OR EDGEPOS(xGR_MAXR_T_EO.Q) THEN	bAdd_CBearing_Hi_Offset	:= TRUE; 	END_IF

	FOR iCntCB:= 1 TO xEngType.NumberOfCylinder BY 1 DO

		IF  NOT Para.bT_CBearing_Exist 									OR
			(VIS2MM.bDem_T_CBearing_Calib AND (iNumCB_Calib = 0 	OR	 		(* all cylinders gets calibrated *)
									   		   iNumCB_Calib = iCntCB  ))
		THEN
			bErrCBTemp_Ms[iCntCB]			:= FALSE;
			bErrCBTemp_Hi[iCntCB]			:= FALSE;
			bErrCBTemp_HiHi[iCntCB]			:= FALSE;
			bErrCBTempMDev_Lo[iCntCB]		:= FALSE;
			bErrCBTempMDev_HiHi[iCntCB]		:= FALSE;
			bErrCBTempSig_Lo[iCntCB] 		:= FALSE;
			xTON_MsDelay[iCntCB](IN			:= FALSE);
		ELSE
			(* MEASUREMENT ERROR *)
			xTON_MsDelay[iCntCB](IN			:= rT_CBearing[iCntCB] <= 5 AND xTON_ReleaseMon.Q,
								 PT			:= T#45s);

			bErrCBTemp_Ms[iCntCB]			:= xTON_MsDelay[iCntCB].Q;

			(* MAXIMUM WARNING / ERROR *)
			IF IN_EG.rP_Act_Norm > 0.3 THEN
				(* Leistung >  30% Nennleistung *)
				bErrCBTemp_Hi[iCntCB]		:= rT_CBearing[iCntCB] > Para.rT_CBearing_Hi;
				bErrCBTemp_HiHi[iCntCB] 	:= rT_CBearing[iCntCB] > Para.rT_CBearing_HiHi;
			ELSE
				(* Leistung <= 30% Nennleistung -->   offset *)
				IF bAdd_CBearing_Hi_Offset	THEN
					(* Oil temperature > 65°C  --> + offset *)
					bErrCBTemp_Hi[iCntCB]	:= rT_CBearing[iCntCB] > Para.rT_CBearing_Hi   + Para.rT_CBearing_Hi_Offset;
					bErrCBTemp_HiHi[iCntCB]	:= rT_CBearing[iCntCB] > Para.rT_CBearing_HiHi + Para.rT_CBearing_Hi_Offset;
				ELSE
					(* Oil temperature < 65°C  --> - offset *)
					bErrCBTemp_Hi[iCntCB]	:= rT_CBearing[iCntCB] > Para.rT_CBearing_Hi   - Para.rT_CBearing_Hi_Offset;
					bErrCBTemp_HiHi[iCntCB]	:= rT_CBearing[iCntCB] > Para.rT_CBearing_HiHi - Para.rT_CBearing_Hi_Offset;
				END_IF
			END_IF

			(* MEDIAN DEVIATION *)
			bErrCBTempMDev_Lo[iCntCB]		:= (rT_CBearing[iCntCB] < xMEDIAN_Temp.median - Para.rT_CBearing_MDev_HiHi) AND
									 		   (rT_CBearing[iCntCB] > 5);

			bErrCBTempMDev_HiHi[iCntCB]		:= (rT_CBearing[iCntCB] > xMEDIAN_Temp.median + Para.rT_CBearing_MDev_HiHi) AND
									 		   (rT_CBearing[iCntCB] > 5);

			(* SIGNAL STRENGTH ERROR *)
			bErrCBTempSig_Lo[iCntCB] 		:= MM2VIS.iPc_T_CBearing_Sig[iCntCB] < Para.iPc_T_CBearing_Sig_Lo;
		END_IF
	END_FOR

	(********************************************************************************************************************************)
	(************************              				 AMM sequencer	 		             	           **************************)
	(********************************************************************************************************************************)
	xTON_SecondTick(IN := NOT xTON_SecondTick.Q, 					PT:= T#800ms);					(* 800ms + 2x cycle time = 1 sec.*)
	xTON_ReleaseMon(IN := IN_EG.rN_EngAct > 400, 					PT:= T#60s);					(* monitoring delay *)
	xTON_ReleaseMon1(IN:= IN_EG.rN_EngAct >= Para.rN_EngNom * 0.95, PT:= T#60s);					(* monitoring delay *)

	(* ERROR   conrod bearing temperature measuring signal failure *)
	xAmmSeq_TempMs.Enable				:= NOT IN_EG.tAB2EG.bResetWarning;
	xAmmSeq_TempMs.ClockPulse			:= xTON_SecondTick.Q;
	xAmmSeq_TempMs.NrOfBits				:= 25;
	xAmmSeq_TempMs.BitArray				:= ADR(bErrCBTemp_Ms);
	xAmmSeq_TempMs();

	bAMM_T_CBearing_Ms					:= xAmmSeq_TempMs.Alarm1;															(* W2790 *)
	bOpM_T_CBearing_Ms					:= xAmmSeq_TempMs.Alarm2;															(* B2806 *)
	iNum_T_CBearing_Ms  				:= xAmmSeq_TempMs.ErrorNr;

	MM2VIS.iOpM_Pc_T_CBearing_Sig		:= MM2VIS.iPc_T_CBearing_Sig[iNum_T_CBearing_Ms]; 	(* signal strength of tripped cylinder *)

	(* WARNING conrod bearing temperature maximum  *)
	xAmmSeq_TempHi.Enable				:= NOT IN_EG.tAB2EG.bResetWarning AND bOMSS_MAT;
	xAmmSeq_TempHi.ClockPulse			:= xTON_SecondTick.Q;
	xAmmSeq_TempHi.NrOfBits				:= 25;
	xAmmSeq_TempHi.BitArray				:= ADR(bErrCBTemp_Hi);
	xAmmSeq_TempHi();

	bAMM_T_CBearing_Hi					:= xAmmSeq_TempHi.Alarm1 	OR IN_EG.tT_CBearing_Hi.Di;								(* W2544 *)
	bOpM_T_CBearing_Hi					:= xAmmSeq_TempHi.Alarm2;															(* B2807 *)
	iNum_T_CBearing_Hi  				:= xAmmSeq_TempHi.ErrorNr;

	(* ERROR   conrod bearing temperature maximum  *)
	xAmmSeq_TempHiHi.Enable				:= NOT IN_EG.tAB2EG.bResetTrip AND bOMSS_MAT;
	xAmmSeq_TempHiHi.ClockPulse			:= xTON_SecondTick.Q;
	xAmmSeq_TempHiHi.NrOfBits			:= 25;
	xAmmSeq_TempHiHi.BitArray			:= ADR(bErrCBTemp_HiHi);
	xAmmSeq_TempHiHi();

	bAMM_T_CBearing_HiHi				:= xAmmSeq_TempHiHi.Alarm1	OR IN_EG.tT_CBearing_HiHi.Di;							(* A2230 *)

	(* ERROR   conrod bearing temperature - negative MEDIAN deviation maximum  *)
	xAmmSeq_TempMDevLo.Enable			:= NOT IN_EG.tAB2EG.bResetWarning AND xTON_ReleaseMon.Q;
	xAmmSeq_TempMDevLo.ClockPulse		:= xTON_SecondTick.Q;
	xAmmSeq_TempMDevLo.NrOfBits			:= 25;
	xAmmSeq_TempMDevLo.BitArray			:= ADR(bErrCBTempMDev_Lo);
	xAmmSeq_TempMDevLo();

	bAMM_T_CBearing_MDev_Lo				:= xAmmSeq_TempMDevLo.Alarm1;														(* W9219 *)
	bOpM_T_CBearing_MDev_Lo				:= xAmmSeq_TempMDevLo.Alarm2;														(* B2959 *)
	iNum_T_CBearing_MDev_Lo				:= xAmmSeq_TempMDevLo.ErrorNr;

	(* ERROR   conrod bearing temperature - positive MEDIAN deviation maximum  *)
	xAmmSeq_TempMDevHiHi.Enable			:= NOT (IN_EG.tAB2EG.bResetTrip OR (IN_EG.tAB2EG.bResetWarning AND bMsg2286_Test)) AND
										   xTON_ReleaseMon.Q;
	xAmmSeq_TempMDevHiHi.ClockPulse		:= xTON_SecondTick.Q;
	xAmmSeq_TempMDevHiHi.NrOfBits		:= 25;
	xAmmSeq_TempMDevHiHi.BitArray		:= ADR(bErrCBTempMDev_HiHi);
	xAmmSeq_TempMDevHiHi();

	bAMM_T_CBearing_MDev_HiHi			:= xAmmSeq_TempMDevHiHi.Alarm1;														(* A2286 *)
	bOpM_T_CBearing_MDev_HiHi			:= xAmmSeq_TempMDevHiHi.Alarm2;														(* B2905 *)
	iNum_T_CBearing_MDev_HiHi			:= xAmmSeq_TempMDevHiHi.ErrorNr;

	(* ERROR   conrod bearing signal intensity minimum  *)
	xAmmSeq_TempSigLo.Enable			:= NOT IN_EG.tAB2EG.bResetWarning AND xTON_ReleaseMon1.Q AND iSt_ReadStrength = 0;
	xAmmSeq_TempSigLo.ClockPulse		:= xTON_SecondTick.Q;
	xAmmSeq_TempSigLo.NrOfBits			:= 25;
	xAmmSeq_TempSigLo.BitArray			:= ADR(bErrCBTempSig_Lo);
	xAmmSeq_TempSigLo();

	bAMM_T_CBearing_Sig_Lo				:= xAmmSeq_TempSigLo.Alarm1;														(* W3559 *)
	bOpM_T_CBearing_Sig_Lo				:= xAmmSeq_TempSigLo.Alarm2;														(* B2822 *)
	iNum_T_CBearing_Sig_Lo  			:= xAmmSeq_TempSigLo.ErrorNr;

	(********************************************************************************************************************************)
	(************************              						VISU	 	             	   	        	*************************)
	(********************************************************************************************************************************)
	IF iCntCB_MsOk > 0 THEN
		MM2VIS.rT_CBearing_Min			:= rT_CBearing_Min;
		MM2VIS.rT_CBearing_Max			:= rT_CBearing_Max;
		MM2VIS.rT_CBearing_Avg			:= rT_CBearing_Sum / INT_TO_REAL(iCntCB_MsOk);
	ELSE
		MM2VIS.rT_CBearing_Min			:= 0;
		MM2VIS.rT_CBearing_Max			:= 0;
		MM2VIS.rT_CBearing_Min			:= 0;
	END_IF

	IF xEngType.NumberOfCylinder > 0 THEN
		MM2VIS.iPc_T_CBearing_Sig_Min	:= iPc_T_CBearing_Sig_Min;
		MM2VIS.iPc_T_CBearing_Sig_Max	:= iPc_T_CBearing_Sig_Max;
		MM2VIS.iPc_T_CBearing_Sig_Avg	:= iPc_T_CBearing_Sig_Sum  / USINT_TO_INT(xEngType.NumberOfCylinder);

		MM2VIS.iPc_T_CBearing_Gain_Min	:= iPc_T_CBearing_Gain_Min;
		MM2VIS.iPc_T_CBearing_Gain_Max	:= iPc_T_CBearing_Gain_Max;
		MM2VIS.iPc_T_CBearing_Gain_Avg	:= iPc_T_CBearing_Gain_Sum / USINT_TO_INT(xEngType.NumberOfCylinder);
	ELSE
		MM2VIS.iPc_T_CBearing_Sig_Min	:= 0;
		MM2VIS.iPc_T_CBearing_Sig_Max	:= 0;
		MM2VIS.iPc_T_CBearing_Sig_Avg	:= 0;
		MM2VIS.iPc_T_CBearing_Gain_Min	:= 0;
		MM2VIS.iPc_T_CBearing_Gain_Max	:= 0;
		MM2VIS.iPc_T_CBearing_Gain_Avg	:= 0;
	END_IF

	(* bearing position (number) for operating message *)
	MM2VIS.iNum_T_CBearing_MsMs			:= iNum_T_CBearing_Ms;
	MM2VIS.iNum_T_CBearing_Hi			:= iNum_T_CBearing_Hi;
	MM2VIS.iNum_T_CBearing_Sig_Lo		:= iNum_T_CBearing_Sig_Lo;
	MM2VIS.iNum_T_CBearing_MDev_Lo		:= iNum_T_CBearing_MDev_Lo;
	MM2VIS.iNum_T_CBearing_MDev_HiHi	:= iNum_T_CBearing_MDev_HiHi;
END_PROGRAM
```

#### ConRoMonInit.st - Initialization code
```iecst
(*******************************************************************************
ConRoMon: Conrod bearing temperature CANopen Sensor (init)

This code is confidential AND proprietary to the INNIO Company.
It may NOT be used in any form, or reproduced in any manner, without the express
written permission of the INNIO Company.
Copyright, INNIO Company, 2019

Customized modifications: -
------------------------

History:
-------
V0.1	27-05-2009	Kröll,Waldhart,Weigl generated
V0.11	22-03-2010	Waldhart,  enhanced FOR 24 cylinder
V0.13	27.03.2013	Tinello, restructured FOR modular SW
V0.14	14.01.2015	Tinello	 restructured FOR XT4

Instructions FOR use:
--------------------

Outstandings:
------------
*******************************************************************************)
PROGRAM _INIT

	(* send parameters to kongsberg system *)
	iCnt_Para				:= 0;
	iSt_Para				:= 0;
	iCntCB_Para				:= 1;

END_PROGRAM
```

#### ConRoMon.typ - Local data types
```iecst
TYPE
	_ConRodMon : 	STRUCT
		Address : USINT;
		IndexLo : USINT;
		IndexHi : USINT;
		Cylinder : USINT;
		Data : INT;
		Unused : INT;
	END_STRUCT;
	_CBearing_Sig : 	STRUCT
		Act : ARRAY[0..10]OF INT;
	END_STRUCT;
END_TYPE
```

#### ConRoMon.var - Local variables
```iecst
VAR
	bAdd_CBearing_Hi_Offset : BOOL := FALSE; (*TRUE = add conrod bearing temperature maximum - offset *)
	bCalib_Again : ARRAY[0..24] OF BOOL := [25(FALSE)]; (*TRUE = calibrate again*)
	bErrCBTempMDev_HiHi : ARRAY[0..24] OF BOOL := [25(FALSE)]; (*conrod bearing temperature - positive deviation from Median - maximum error*)
	bErrCBTempMDev_Lo : ARRAY[0..24] OF BOOL := [25(FALSE)]; (*conrod bearing temperature - negative deviation from Median - maximum error*)
	bErrCBTempSig_Lo : ARRAY[0..24] OF BOOL := [25(FALSE)]; (*conrod bearing signal intensity - minimum error*)
	bErrCBTemp_Hi : ARRAY[0..24] OF BOOL := [25(FALSE)]; (*conrod bearing temperature - maximum warning*)
	bErrCBTemp_HiHi : ARRAY[0..24] OF BOOL := [25(FALSE)]; (*conrod bearing temperature - maximum error *)
	bErrCBTemp_Ms : ARRAY[0..24] OF BOOL := [25(FALSE)]; (*conrod bearing temperature - measurement signal failure *)
	bQueueInitDone : BOOL := FALSE; (*for init*)
	bReadStrength : BOOL := FALSE; (*TRUE = Read signal strength of conrod bearing temperature*)
	bRel_CBearing_CAN : BOOL := FALSE; (*conrod bearing CAN bus released for read and write*)
	bWrongCylinder : BOOL := FALSE; (*error bit - wrong cylinder information*)
	DATA_R : _ConRodMon := (0); (*confirmation of written parameter/commands to kongsberg system - SDO*)
	DATA_W : _ConRodMon := (0); (*write parameter/commands to kongsberg system - SDO*)
	i : USINT := 1; (*counter for cylinder number*)
	iCntCB : USINT := 0; (*counter for conrod bearing number*)
	iCntCB_Calib : USINT := 1; (*counter for cylinder number*)
	iCntCB_MsOk : USINT := 0; (*counter for conrod bearings without measurement signal error*)
	iCntCB_Para : USINT := 1; (*counter for cylinder number*)
	iCntCB_Read : USINT := 1; (*counter for cylinder number*)
	iCntCB_ReadAct : USINT := 1; (*counter for strength average*)
	iCnt_Para : INT := 0; (*counter for parameter*)
	ii : USINT := 1; (*counter for average*)
	iNumCalib_Again : USINT := 0; (*Cylinder number to calibrate again*)
	iNumCB_Calib : USINT := 0; (*SAVE - conrod bearing position (number) to calibrate [0 = all]*)
	iNum_T_CBearing_Hi : USINT := 0; (*conrod bearing temperature maximum - bearing position (number)*)
	iNum_T_CBearing_MDev_HiHi : USINT := 0; (*conrod bearing temperature - positive deviation from MEDIAN maximum - bearing position (number)*)
	iNum_T_CBearing_MDev_Lo : USINT := 0; (*conrod bearing temperature - negative deviation from MEDIAN maximum - bearing position (number)*)
	iNum_T_CBearing_Ms : USINT := 0; (*conrod bearing temperature measurement signal failure - bearing position (number)*)
	iNum_T_CBearing_Sig_Lo : USINT := 0; (*conrod bearing signal intensity minimum - bearing position (number)*)
	iPc_T_CBearing_Gain_Act : ARRAY[0..24] OF _CBearing_Sig := [25(0)]; (*actual receiver gain level from conrod bearing temperature sensor [%]*)
	iPc_T_CBearing_Gain_ActSum : INT := 0; (*sum of actual receiver gain level from conrod bearing temperature sensor [%]*)
	iPc_T_CBearing_Gain_Max : INT := 0; (*maximum receiver gain level from conrod bearing temperature sensor [%]*)
	iPc_T_CBearing_Gain_Min : INT := 0; (*minimum receiver gain level from conrod bearing temperature sensor [%]*)
	iPc_T_CBearing_Gain_Sum : INT := 0; (*sum of receiver gain level from conrod bearing temperature sensor [%]*)
	iPc_T_CBearing_Sig_Act : ARRAY[0..24] OF _CBearing_Sig := [25(0)]; (*actual signal strength from conrod bearing temperature sensor [%]*)
	iPc_T_CBearing_Sig_ActSum : INT := 0; (*sum of actual signal strength from conrod bearing temperature sensor [%]*)
	iPc_T_CBearing_Sig_Max : INT := 0; (*maximum signal strength from conrod bearing temperature [%]*)
	iPc_T_CBearing_Sig_Min : INT := 0; (*minimum signal strength from conrod bearing temperature [%]*)
	iPc_T_CBearing_Sig_Sum : INT := 0; (*sum of signal strength from conrod bearing temperature sensor [%]*)
	iSt_Calib : INT := 0; (*State - calibration*)
	iSt_Para : INT := 0; (*State - parameter writing*)
	iSt_ReadGain : INT := 0; (*State - receiver gain level*)
	iSt_ReadStrength : INT := 0; (*State - signal strength*)
	rT_CBearing : ARRAY[0..24] OF REAL; (*conrod bearing temperature [°C]*) (* *) (*V04.02.00.00*)
	rT_CBearing_Max : REAL := 0.0; (*maximal conrod bearing temperature*)
	rT_CBearing_Min : REAL := 0.0; (*minimal conrod bearing temperature*)
	rT_CBearing_Sum : REAL := 0.0; (*actual sum of all conrod bearing temperatures*)
	TEMP : _ConRodMon := (0); (*conrod bearing temperature from kongsberg-System - PDO's*)
	xAmmSeq_TempHi : AmmSequence := (0); (*FuB*)
	xAmmSeq_TempHiHi : AmmSequence := (0); (*FuB*)
	xAmmSeq_TempMDevHiHi : AmmSequence := (0); (*FuB*)
	xAmmSeq_TempMDevLo : AmmSequence := (0); (*FuB*)
	xAmmSeq_TempMs : AmmSequence := (0); (*FuB*)
	xAmmSeq_TempSigLo : AmmSequence := (0); (*FuB*)
	xCANqueue_CB_Temp : CANqueue := (0); (*FuB*)
	xCANrd_CB_Temp : CANrd := (0); (*FuB*)
	xCANread_CB_Data : CANread := (0); (*FuB*)
	xCANwrite_CB_Data : CANwrite := (0); (*FuB*)
	xGR_MAXR_T_EO : GR_MAXR := (0); (*FuB*)
	xGR_MINR_T_EO : GR_MINR := (0); (*FuB*)
	xMEDIAN_Temp : RMEDIAN24 := (0); (*FuB*)
	xTON_Calibration : TON := (0); (*FuB*)
	xTON_CANopen : TON := (0); (*FuB*)
	xTON_CANread : TON := (0); (*FuB*)
	xTON_MsDelay : ARRAY[0..24] OF TON := [25((0))]; (*FuB*)
	xTON_ParaSet : TON := (0); (*FuB*)
	xTON_ReadStrength : TON := (0); (*FuB*)
	xTON_ReleaseMon : TON := (0); (*FuB*)
	xTON_ReleaseMon1 : TON := (0); (*FuB*)
	xTON_SecondTick : TON := (0); (*FuB*)
	xTON_WriteAck : TON := (0); (*FuB*)
	xTON_WriteMax : TON := (0); (*FuB*)
END_VAR
```

### Program Logical/EngineGeneral/IdleFric (IEC, version 4.10.0) - Idle Friction Monitoring

#### IdleFricCyclic.st - Cyclic code
```iecst
(*******************************************************************************
MainBearing: idle friction monitoring (cyclic)

This code is confidential AND proprietary to the INNIO Company.
It may NOT be used in any form, or reproduced in any manner, without the express
written permission of the INNIO Company.
Copyright, INNIO Company, 2021

- check throttle position, boost pressure and speed to prevent engine damage

Customized modifications: -
------------------------

History:
-------
V4.4	28-01-2016	Weitzer, 	generated
		05-12-2016	Weitzer, 	add activation with service button for 10 op hours
V4.4.1	07-03-2017	Weitzer,	correct funktion according to spec
V4.4.2	19-07-2017	Weitzer,    change boost pressure limit to 0.70 bar
V4.10	27.01.2021	Tinello,  	BugFix: Timer-FuB's

Instructions FOR use:
--------------------

Outstandings:
------------

*******************************************************************************)
PROGRAM _CYCLIC

	(* activation of function *)

	(* activate monitoring with service button *)
	IF Para.bIdleFrictionMon THEN

		(* increase counter *)
		iCntOpH := MIN(iCntOpH + BOOL_TO_UINT(EDGEPOS(IN_EG.tImp_OpHour.Do)), 10000);
		(* counter reset *)
		IF EDGEPOS(IN_EG.bServiceMode) THEN
			iCntOpH := 0;
		END_IF;

		bServiceMon := iCntOpH <= 10;
	ELSE
		bServiceMon := FALSE;
	END_IF;

	(* service button was activated within the last 10 operating hours *)
	IF bServiceMon THEN

		(* activate monitoring *)

//		bMonitoringAct :=	(IN_EG.rN_EngAct > (Para.rN_EngNom - rN_Hys) AND IN_EG.rP_Act_Norm < 0.01)  OR
//							(xTON_Monitoring.Q AND (IN_EG.tEng_Run.Do AND NOT IN_EG.tGCB_On.Di));
//
//		xTON_Monitoring.IN := bMonitoringAct;
//		xTON_Monitoring.PT := T#5s;
//		xTON_Monitoring;
//
//
//		(* monitoring *)
//
//		IF bMonitoringAct THEN
//			IF IN_EG.rPos_TV < rPos_TV_HiHi OR xTON_Monitoring.Q THEN
//				IF IN_EG.rPos_TV >= rPos_TV_HiHi OR IN_EG.rPr_Ch_P2s_Avg > rPr_Ch_P2s_HiHi OR IN_EG.rN_EngAct < (Para.rN_EngNom - rN_Hys) THEN
//					bAMM_IdleFriction_HiHi := TRUE;
//				END_IF;
//			END_IF;
//		ELSE
//			bAMM_IdleFriction_HiHi := FALSE;
//		END_IF;

		(* activate monitoring *)

		xTON_Monitoring.IN := IN_EG.rN_EngAct > (Para.rN_EngNom - rN_Hys) AND IN_EG.rP_Act_Norm < 0.01 AND IN_EG.tEng_Run.Do AND NOT IN_EG.tGCB_On.Di;
		xTON_Monitoring.PT := T#8s;
		xTON_Monitoring;

		bMonitoringAct := 	xTON_Monitoring.Q OR
							(
								IN_EG.rN_EngAct > (Para.rN_EngNom - rN_Hys)
							AND IN_EG.rP_Act_Norm < 0.01 AND IN_EG.tEng_Run.Do AND NOT IN_EG.tGCB_On.Di
							AND IN_EG.rPos_TV < rPos_TV_HiHi
							AND IN_EG.rPr_Ch_P2s_Avg < rPr_Ch_P2s_HiHi
							);

		(* monitoring *)

		IF bMonitoringAct THEN
			IF IN_EG.rPos_TV >= rPos_TV_HiHi OR IN_EG.rPr_Ch_P2s_Avg > rPr_Ch_P2s_HiHi OR IN_EG.rN_EngAct < (Para.rN_EngNom - rN_Hys) THEN
				bAMM_IdleFriction_HiHi := TRUE;
			END_IF;
		ELSE
			bAMM_IdleFriction_HiHi := FALSE;
		END_IF;

	ELSE
		bAMM_IdleFriction_HiHi := FALSE;
		xTON_Monitoring(IN	   := FALSE);
	END_IF;

END_PROGRAM
```

#### IdleFricInit.st - Initialization code
```iecst
(*******************************************************************************
MainBearing: idle friction monitoring (init)

This code is confidential AND proprietary to the INNIO Company.
It may NOT be used in any form, or reproduced in any manner, without the express
written permission of the INNIO Company.
Copyright, INNIO Company, 2019

- check throttle position, boost pressure AND speed TO prevent engine damage

Customized modifications: -
------------------------

History:
-------
V4.4	28-01-2016	Weitzer, 	generated
V4.4.2	19-07-2017	Weitzer,    change boost pressure limit to 0.70 bar

Instructions FOR use:
--------------------

Outstandings:
------------

*******************************************************************************)

PROGRAM _INIT

	(* define limits *)
	rN_Hys 			:= 20.0;	(* speed *)
	rPos_TV_HiHi	:= 0.15;	(* throttle valve position *)
	rPr_Ch_P2s_HiHi := 0.70;	(* boost pressure *)

	(* deactivate function after restart of the PLC system *)
	IF iCntOpH = 0 THEN
		iCntOpH := 11;
	END_IF;

END_PROGRAM
```

#### IdleFric.var - Local variables
```iecst
VAR
	bMonitoringAct : BOOL := FALSE; (*Monitoring active*)
	rN_Hys : REAL := 0; (*speed hysteresis*)
	rPos_TV_HiHi : REAL := 0; (*throttle valve position maximum*)
	rPr_Ch_P2s_HiHi : REAL := 0; (*boost pressure maximum*)
	xTON_Monitoring : TON := (0); (*FuB*)
	iCntOpH : UINT;
	bServiceMon : BOOL := 0;
END_VAR
```

### Program Logical/EngineGeneral/MsgEG (IEC, version 4.25.0) - Alarms generation
